	X =  49.000  mm,	Y =  112.000  mm,	Z =   -1.000 mm,
	W =-180.000 deg,	P =   0.000 deg,	R =    90.000 deg
};
P[5913]{
   GP1:
	UF : 1, UT : 4,		CONFIG : 'N U T, 0, 0, 0',
	X =  49.000  mm,	Y =  112.000  mm,	Z =   15.000 mm,
	W =-180.000 deg,	P =   0.000 deg,	R =    90.000 deg
};
P[5992]{
   GP1:
	UF : 1, UT : 4,		CONFIG : 'N U T, 0, 0, 0',
	X =  43.000  mm,	Y =  115.000  mm,	Z =   15.000 mm,
	W =-180.000 deg,	P =   0.000 deg,	R =    90.000 deg
};
P[5993]{
   GP1:
	UF : 1, UT : 4,		CONFIG : 'N U T, 0, 0, 0',
	X =  43.000  mm,	Y =  115.000  mm,	Z =   -1.000 mm,
	W =-180.000 deg,	P =   0.000 deg,	R =    90.000 deg
};
P[5994]{
   GP1:
	UF : 1, UT : 4,		CONFIG : 'N U T, 0, 0, 0',
	X =  43.000  mm,	Y =  115.000  mm,	Z =   15.000 mm,
	W =-180.000 deg,	P =   0.000 deg,	R =    90.000 deg
};
P[5995]{
   GP1:
	UF : 1, UT : 4,		CONFIG : 'N U T, 0, 0, 0',
	X =  46.000  mm,	Y =  115.000  mm,	Z =   15.000 mm,
	W =-180.000 deg,	P =   0.000 deg,	R =    90.000 deg
};
P[5996]{
   GP1:
	UF : 1, UT : 4,		CONFIG : 'N U T, 0, 0, 0',
	X =  46.000  mm,	Y =  115.000  mm,	Z =   -1.000 mm,
	W =-180.000 deg,	P =   0.000 deg,	R =    90.000 deg
};
P[5997]{
   GP1:
	UF : 1, UT : 4,		CONFIG : 'N U T, 0, 0, 0',
	X =  46.000  mm,	Y =  115.000  mm,	Z =   15.000 mm,
	W =-180.000 deg,	P =   0.000 deg,	R =    90.000 deg
};
P[5998]{
   GP1:
	UF : 1, UT : 4,		CONFIG : 'N U T, 0, 0, 0',
	X =  49.000  mm,	Y =  115.000  mm,	Z =   15.000 mm,
	W =-180.000 deg,	P =   0.000 deg,	R =    90.000 deg
};
P[5999]{
   GP1:
	UF : 1, UT : 4,		CONFIG : 'N U T, 0, 0, 0',
	X =  49.000  mm,	Y =  115.000  mm,	Z =   -1.000 mm,
	W =-180.000 deg,	P =   0.000 deg,	R =    90.000 deg
};
P[6000]{
   GP1:
	UF : 1, UT : 4,		CONFIG : 'N U T, 0, 0, 0',
	X =  49.000  mm,	Y =  115.000  mm,	Z =   15.000 mm,
	W =-180.000 deg,	P =   0.000 deg,	R =    90.000 deg
};
P[6001]{
   GP1:
	UF : 1, UT : 4,		CONFIG : 'N U T, 0, 0, 0',
	X =  52.000  mm,	Y =  115.000  mm,	Z =   15.000 mm,
	W =-180.000 deg,	P =   0.000 deg,	R =    90.000 deg
};
P[6002]{
   GP1:
	UF : 1, UT : 4,		CONFIG : 'N U T, 0, 0, 0',
	X =  52.000  mm,	Y =  115.000  mm,	Z =   -1.000 mm,
	W =-180.000 deg,	P =   0.000 deg,	R =    90.000 deg
};
P[6003]{
   GP1:
	UF : 1, UT : 4,		CONFIG : 'N U T, 0, 0, 0',
	X =  52.000  mm,	Y =  115.000  mm,	Z =   15.000 mm,
	W =-180.000 deg,	P =   0.000 deg,	R =    90.000 deg
};
P[6004]{
   GP1:
	UF : 1, UT : 4,		CONFIG : 'N U T, 0, 0, 0',
	X =  55.000  mm,	Y =  115.000  mm,	Z =   15.000 mm,
	W =-180.000 deg,	P =   0.000 deg,	R =    90.000 deg
};
P[6005]{
   GP1:
	UF : 1, UT : 4,		CONFIG : 'N U T, 0, 0, 0',
	X =  55.000  mm,	Y =  115.000  mm,	Z =   -1.000 mm,
	W =-180.000 deg,	P =   0.000 deg,	R =    90.000 deg
};
P[6006]{
   GP1:
	UF : 1, UT : 4,		CONFIG : 'N U T, 0, 0, 0',
	X =  55.000  mm,	Y =  115.000  mm,	Z =   15.000 mm,
	W =-180.000 deg,	P =   0.000 deg,	R =    90.000 deg
};
P[6007]{
   GP1:
	UF : 1, UT : 4,		CONFIG : 'N U T, 0, 0, 0',
	X =  58.000  mm,	Y =  115.000  mm,	Z =   15.000 mm,
	W =-180.000 deg,	P =   0.000 deg,	R =    90.000 deg
};
P[6008]{
   GP1:
	UF : 1, UT : 4,		CONFIG : 'N U T, 0, 0, 0',
	X =  58.000  mm,	Y =  115.000  mm,	Z =   -1.000 mm,
	W =-180.000 deg,	P =   0.000 deg,	R =    90.000 deg
};
P[6009]{
   GP1:
	UF : 1, UT : 4,		CONFIG : 'N U T, 0, 0, 0',
	X =  58.000  mm,	Y =  115.000  mm,	Z =   15.000 mm,
	W =-180.000 deg,	P =   0.000 deg,	R =    90.000 deg
};
P[6010]{
   GP1:
	UF : 1, UT : 4,		CONFIG : 'N U T, 0, 0, 0',
	X =  103.000  mm,	Y =  115.000  mm,	Z =   15.000 mm,
	W =-180.000 deg,	P =   0.000 deg,	R =    90.000 deg
};
P[6011]{
   GP1:
	UF : 1, UT : 4,		CONFIG : 'N U T, 0, 0, 0',
	X =  103.000  mm,	Y =  115.000  mm,	Z =   -1.000 mm,
	W =-180.000 deg,	P =   0.000 deg,	R =    90.000 deg
};
P[6012]{
   GP1:
	UF : 1, UT : 4,		CONFIG : 'N U T, 0, 0, 0',
	X =  103.000  mm,	Y =  115.000  mm,	Z =   15.000 mm,
	W =-180.000 deg,	P =   0.000 deg,	R =    90.000 deg
};
P[6058]{
   GP1:
	UF : 1, UT : 4,		CONFIG : 'N U T, 0, 0, 0',
	X =  16.000  mm,	Y =  118.000  mm,	Z =   15.000 mm,
	W =-180.000 deg,	P =   0.000 deg,	R =    90.000 deg
};
P[6059]{
   GP1:
	UF : 1, UT : 4,		CONFIG : 'N U T, 0, 0, 0',
	X =  16.000  mm,	Y =  118.000  mm,	Z =   -1.000 mm,
	W =-180.000 deg,	P =   0.000 deg,	R =    90.000 deg
};
P[6060]{
   GP1:
	UF : 1, UT : 4,		CONFIG : 'N U T, 0, 0, 0',
	X =  16.000  mm,	Y =  118.000  mm,	Z =   15.000 mm,
	W =-180.000 deg,	P =   0.000 deg,	R =    90.000 deg
};
P[6061]{
   GP1:
	UF : 1, UT : 4,		CONFIG : 'N U T, 0, 0, 0',
	X =  19.000  mm,	Y =  118.000  mm,	Z =   15.000 mm,
	W =-180.000 deg,	P =   0.000 deg,	R =    90.000 deg
};
P[6062]{
   GP1:
	UF : 1, UT : 4,		CONFIG : 'N U T, 0, 0, 0',
	X =  19.000  mm,	Y =  118.000  mm,	Z =   -1.000 mm,
	W =-180.000 deg,	P =   0.000 deg,	R =    90.000 deg
};
P[6063]{
   GP1:
	UF : 1, UT : 4,		CONFIG : 'N U T, 0, 0, 0',
	X =  19.000  mm,	Y =  118.000  mm,	Z =   15.000 mm,
	W =-180.000 deg,	P =   0.000 deg,	R =    90.000 deg
};
P[6070]{
   GP1:
	UF : 1, UT : 4,		CONFIG : 'N U T, 0, 0, 0',
	X =  28.000  mm,	Y =  118.000  mm,	Z =   15.000 mm,
	W =-180.000 deg,	P =   0.000 deg,	R =    90.000 deg
};
P[6071]{
   GP1:
	UF : 1, UT : 4,		CONFIG : 'N U T, 0, 0, 0',
	X =  28.000  mm,	Y =  118.000  mm,	Z =   -1.000 mm,
	W =-180.000 deg,	P =   0.000 deg,	R =    90.000 deg
};
P[6072]{
   GP1:
	UF : 1, UT : 4,		CONFIG : 'N U T, 0, 0, 0',
	X =  28.000  mm,	Y =  118.000  mm,	Z =   15.000 mm,
	W =-180.000 deg,	P =   0.000 deg,	R =    90.000 deg
};
P[6079]{
   GP1:
	UF : 1, UT : 4,		CONFIG : 'N U T, 0, 0, 0',
	X =  37.000  mm,	Y =  118.000  mm,	Z =   15.000 mm,
	W =-180.000 deg,	P =   0.000 deg,	R =    90.000 deg
};
P[6080]{
   GP1:
	UF : 1, UT : 4,		CONFIG : 'N U T, 0, 0, 0',
	X =  37.000  mm,	Y =  118.000  mm,	Z =   -1.000 mm,
	W =-180.000 deg,	P =   0.000 deg,	R =    90.000 deg
};
P[6081]{
   GP1:
	UF : 1, UT : 4,		CONFIG : 'N U T, 0, 0, 0',
	X =  37.000  mm,	Y =  118.000  mm,	Z =   15.000 mm,
	W =-180.000 deg,	P =   0.000 deg,	R =    90.000 deg
};
P[6082]{
   GP1:
	UF : 1, UT : 4,		CONFIG : 'N U T, 0, 0, 0',
	X =  40.000  mm,	Y =  118.000  mm,	Z =   15.000 mm,
	W =-180.000 deg,	P =   0.000 deg,	R =    90.000 deg
};
P[6083]{
   GP1:
	UF : 1, UT : 4,		CONFIG : 'N U T, 0, 0, 0',
	X =  40.000  mm,	Y =  118.000  mm,	Z =   -1.000 mm,
	W =-180.000 deg,	P =   0.000 deg,	R =    90.000 deg
};
P[6084]{
   GP1:
	UF : 1, UT : 4,		CONFIG : 'N U T, 0, 0, 0',
	X =  40.000  mm,	Y =  118.000  mm,	Z =   15.000 mm,
	W =-180.000 deg,	P =   0.000 deg,	R =    90.000 deg
};
P[6085]{
   GP1:
	UF : 1, UT : 4,		CONFIG : 'N U T, 0, 0, 0',
	X =  43.000  mm,	Y =  118.000  mm,	Z =   15.000 mm,
	W =-180.000 deg,	P =   0.000 deg,	R =    90.000 deg
};
P[6086]{
   GP1:
	UF : 1, UT : 4,		CONFIG : 'N U T, 0, 0, 0',
	X =  43.000  mm,	Y =  118.000  mm,	Z =   -1.000 mm,
	W =-180.000 deg,	P =   0.000 deg,	R =    90.000 deg
};
P[6087]{
   GP1:
	UF : 1, UT : 4,		CONFIG : 'N U T, 0, 0, 0',
	X =  43.000  mm,	Y =  118.000  mm,	Z =   15.000 mm,
	W =-180.000 deg,	P =   0.000 deg,	R =    90.000 deg
};
P[6088]{
   GP1:
	UF : 1, UT : 4,		CONFIG : 'N U T, 0, 0, 0',
	X =  46.000  mm,	Y =  118.000  mm,	Z =   15.000 mm,
	W =-180.000 deg,	P =   0.000 deg,	R =    90.000 deg
};
P[6089]{
   GP1:
	UF : 1, UT : 4,		CONFIG : 'N U T, 0, 0, 0',
	X =  46.000  mm,	Y =  118.000  mm,	Z =   -1.000 mm,
	W =-180.000 deg,	P =   0.000 deg,	R =    90.000 deg
};
P[6090]{
   GP1:
	UF : 1, UT : 4,		CONFIG : 'N U T, 0, 0, 0',
	X =  46.000  mm,	Y =  118.000  mm,	Z =   15.000 mm,
	W =-180.000 deg,	P =   0.000 deg,	R =    90.000 deg
};
P[6091]{
   GP1:
	UF : 1, UT : 4,		CONFIG : 'N U T, 0, 0, 0',
	X =  49.000  mm,	Y =  118.000  mm,	Z =   15.000 mm,
	W =-180.000 deg,	P =   0.000 deg,	R =    90.000 deg
};
P[6092]{
   GP1:
	UF : 1, UT : 4,		CONFIG : 'N U T, 0, 0, 0',
	X =  49.000  mm,	Y =  118.000  mm,	Z =   -1.000 mm,
	W =-180.000 deg,	P =   0.000 deg,	R =    90.000 deg
};
P[6093]{
   GP1:
	UF : 1, UT : 4,		CONFIG : 'N U T, 0, 0, 0',
	X =  49.000  mm,	Y =  118.000  mm,	Z =   15.000 mm,
	W =-180.000 deg,	P =   0.000 deg,	R =    90.000 deg
};
P[6094]{
   GP1:
	UF : 1, UT : 4,		CONFIG : 'N U T, 0, 0, 0',
	X =  52.000  mm,	Y =  118.000  mm,	Z =   15.000 mm,
	W =-180.000 deg,	P =   0.000 deg,	R =    90.000 deg
};
P[6095]{
   GP1:
	UF : 1, UT : 4,		CONFIG : 'N U T, 0, 0, 0',
	X =  52.000  mm,	Y =  118.000  mm,	Z =   -1.000 mm,
	W =-180.000 deg,	P =   0.000 deg,	R =    90.000 deg
};
P[6096]{
   GP1:
	UF : 1, UT : 4,		CONFIG : 'N U T, 0, 0, 0',
	X =  52.000  mm,	Y =  118.000  mm,	Z =   15.000 mm,
	W =-180.000 deg,	P =   0.000 deg,	R =    90.000 deg
};
P[6097]{
   GP1:
	UF : 1, UT : 4,		CONFIG : 'N U T, 0, 0, 0',
	X =  55.000  mm,	Y =  118.000  mm,	Z =   15.000 mm,
	W =-180.000 deg,	P =   0.000 deg,	R =    90.000 deg
};
P[6098]{
   GP1:
	UF : 1, UT : 4,		CONFIG : 'N U T, 0, 0, 0',
	X =  55.000  mm,	Y =  118.000  mm,	Z =   -1.000 mm,
	W =-180.000 deg,	P =   0.000 deg,	R =    90.000 deg
};
P[6099]{
   GP1:
	UF : 1, UT : 4,		CONFIG : 'N U T, 0, 0, 0',
	X =  55.000  mm,	Y =  118.000  mm,	Z =   15.000 mm,
	W =-180.000 deg,	P =   0.000 deg,	R =    90.000 deg
};
P[6100]{
   GP1:
	UF : 1, UT : 4,		CONFIG : 'N U T, 0, 0, 0',
	X =  58.000  mm,	Y =  118.000  mm,	Z =   15.000 mm,
	W =-180.000 deg,	P =   0.000 deg,	R =    90.000 deg
};
P[6101]{
   GP1:
	UF : 1, UT : 4,		CONFIG : 'N U T, 0, 0, 0',
	X =  58.000  mm,	Y =  118.000  mm,	Z =   -1.000 mm,
	W =-180.000 deg,	P =   0.000 deg,	R =    90.000 deg
};
P[6102]{
   GP1:
	UF : 1, UT : 4,		CONFIG : 'N U T, 0, 0, 0',
	X =  58.000  mm,	Y =  118.000  mm,	Z =   15.000 mm,
	W =-180.000 deg,	P =   0.000 deg,	R =    90.000 deg
};
P[6133]{
   GP1:
	UF : 1, UT : 4,		CONFIG : 'N U T, 0, 0, 0',
	X =  145.000  mm,	Y =  118.000  mm,	Z =   15.000 mm,
	W =-180.000 deg,	P =   0.000 deg,	R =    90.000 deg
};
P[6134]{
   GP1:
	UF : 1, UT : 4,		CONFIG : 'N U T, 0, 0, 0',
	X =  145.000  mm,	Y =  118.000  mm,	Z =   -1.000 mm,
	W =-180.000 deg,	P =   0.000 deg,	R =    90.000 deg
};
P[6135]{
   GP1:
	UF : 1, UT : 4,		CONFIG : 'N U T, 0, 0, 0',
	X =  145.000  mm,	Y =  118.000  mm,	Z =   15.000 mm,
	W =-180.000 deg,	P =   0.000 deg,	R =    90.000 deg
};
P[6160]{
   GP1:
	UF : 1, UT : 4,		CONFIG : 'N U T, 0, 0, 0',
	X =  16.000  mm,	Y =  121.000  mm,	Z =   15.000 mm,
	W =-180.000 deg,	P =   0.000 deg,	R =    90.000 deg
};
P[6161]{
   GP1:
	UF : 1, UT : 4,		CONFIG : 'N U T, 0, 0, 0',
	X =  16.000  mm,	Y =  121.000  mm,	Z =   -1.000 mm,
	W =-180.000 deg,	P =   0.000 deg,	R =    90.000 deg
};
P[6162]{
   GP1:
	UF : 1, UT : 4,		CONFIG : 'N U T, 0, 0, 0',
	X =  16.000  mm,	Y =  121.000  mm,	Z =   15.000 mm,
	W =-180.000 deg,	P =   0.000 deg,	R =    90.000 deg
};
P[6172]{
   GP1:
	UF : 1, UT : 4,		CONFIG : 'N U T, 0, 0, 0',
	X =  28.000  mm,	Y =  121.000  mm,	Z =   15.000 mm,
	W =-180.000 deg,	P =   0.000 deg,	R =    90.000 deg
};
P[6173]{
   GP1:
	UF : 1, UT : 4,		CONFIG : 'N U T, 0, 0, 0',
	X =  28.000  mm,	Y =  121.000  mm,	Z =   -1.000 mm,
	W =-180.000 deg,	P =   0.000 deg,	R =    90.000 deg
};
P[6174]{
   GP1:
	UF : 1, UT : 4,		CONFIG : 'N U T, 0, 0, 0',
	X =  28.000  mm,	Y =  121.000  mm,	Z =   15.000 mm,
	W =-180.000 deg,	P =   0.000 deg,	R =    90.000 deg
};
P[6187]{
   GP1:
	UF : 1, UT : 4,		CONFIG : 'N U T, 0, 0, 0',
	X =  43.000  mm,	Y =  121.000  mm,	Z =   15.000 mm,
	W =-180.000 deg,	P =   0.000 deg,	R =    90.000 deg
};
P[6188]{
   GP1:
	UF : 1, UT : 4,		CONFIG : 'N U T, 0, 0, 0',
	X =  43.000  mm,	Y =  121.000  mm,	Z =   -1.000 mm,
	W =-180.000 deg,	P =   0.000 deg,	R =    90.000 deg
};
P[6189]{
   GP1:
	UF : 1, UT : 4,		CONFIG : 'N U T, 0, 0, 0',
	X =  43.000  mm,	Y =  121.000  mm,	Z =   15.000 mm,
	W =-180.000 deg,	P =   0.000 deg,	R =    90.000 deg
};
P[6190]{
   GP1:
	UF : 1, UT : 4,		CONFIG : 'N U T, 0, 0, 0',
	X =  46.000  mm,	Y =  121.000  mm,	Z =   15.000 mm,
	W =-180.000 deg,	P =   0.000 deg,	R =    90.000 deg
};
P[6191]{
   GP1:
	UF : 1, UT : 4,		CONFIG : 'N U T, 0, 0, 0',
	X =  46.000  mm,	Y =  121.000  mm,	Z =   -1.000 mm,
	W =-180.000 deg,	P =   0.000 deg,	R =    90.000 deg
};
P[6192]{
   GP1:
	UF : 1, UT : 4,		CONFIG : 'N U T, 0, 0, 0',
	X =  46.000  mm,	Y =  121.000  mm,	Z =   15.000 mm,
	W =-180.000 deg,	P =   0.000 deg,	R =    90.000 deg
};
P[6193]{
   GP1:
	UF : 1, UT : 4,		CONFIG : 'N U T, 0, 0, 0',
	X =  49.000  mm,	Y =  121.000  mm,	Z =   15.000 mm,
	W =-180.000 deg,	P =   0.000 deg,	R =    90.000 deg
};
P[6194]{
   GP1:
	UF : 1, UT : 4,		CONFIG : 'N U T, 0, 0, 0',
	X =  49.000  mm,	Y =  121.000  mm,	Z =   -1.000 mm,
	W =-180.000 deg,	P =   0.000 deg,	R =    90.000 deg
};
P[6195]{
   GP1:
	UF : 1, UT : 4,		CONFIG : 'N U T, 0, 0, 0',
	X =  49.000  mm,	Y =  121.000  mm,	Z =   15.000 mm,
	W =-180.000 deg,	P =   0.000 deg,	R =    90.000 deg
};
P[6196]{
   GP1:
	UF : 1, UT : 4,		CONFIG : 'N U T, 0, 0, 0',
	X =  52.000  mm,	Y =  121.000  mm,	Z =   15.000 mm,
	W =-180.000 deg,	P =   0.000 deg,	R =    90.000 deg
};
P[6197]{
   GP1:
	UF : 1, UT : 4,		CONFIG : 'N U T, 0, 0, 0',
	X =  52.000  mm,	Y =  121.000  mm,	Z =   -1.000 mm,
	W =-180.000 deg,	P =   0.000 deg,	R =    90.000 deg
};
P[6198]{
   GP1:
	UF : 1, UT : 4,		CONFIG : 'N U T, 0, 0, 0',
	X =  52.000  mm,	Y =  121.000  mm,	Z =   15.000 mm,
	W =-180.000 deg,	P =   0.000 deg,	R =    90.000 deg
};
P[6199]{
   GP1:
	UF : 1, UT : 4,		CONFIG : 'N U T, 0, 0, 0',
	X =  55.000  mm,	Y =  121.000  mm,	Z =   15.000 mm,
	W =-180.000 deg,	P =   0.000 deg,	R =    90.000 deg
};
P[6200]{
   GP1:
	UF : 1, UT : 4,		CONFIG : 'N U T, 0, 0, 0',
	X =  55.000  mm,	Y =  121.000  mm,	Z =   -1.000 mm,
	W =-180.000 deg,	P =   0.000 deg,	R =    90.000 deg
};
P[6201]{
   GP1:
	UF : 1, UT : 4,		CONFIG : 'N U T, 0, 0, 0',
	X =  55.000  mm,	Y =  121.000  mm,	Z =   15.000 mm,
	W =-180.000 deg,	P =   0.000 deg,	R =    90.000 deg
};
P[6202]{
   GP1:
	UF : 1, UT : 4,		CONFIG : 'N U T, 0, 0, 0',
	X =  58.000  mm,	Y =  121.000  mm,	Z =   15.000 mm,
	W =-180.000 deg,	P =   0.000 deg,	R =    90.000 deg
};
P[6203]{
   GP1:
	UF : 1, UT : 4,		CONFIG : 'N U T, 0, 0, 0',
	X =  58.000  mm,	Y =  121.000  mm,	Z =   -1.000 mm,
	W =-180.000 deg,	P =   0.000 deg,	R =    90.000 deg
};
P[6204]{
   GP1:
	UF : 1, UT : 4,		CONFIG : 'N U T, 0, 0, 0',
	X =  58.000  mm,	Y =  121.000  mm,	Z =   15.000 mm,
	W =-180.000 deg,	P =   0.000 deg,	R =    90.000 deg
};
P[6205]{
   GP1:
	UF : 1, UT : 4,		CONFIG : 'N U T, 0, 0, 0',
	X =  61.000  mm,	Y =  121.000  mm,	Z =   15.000 mm,
	W =-180.000 deg,	P =   0.000 deg,	R =    90.000 deg
};
P[6206]{
   GP1:
	UF : 1, UT : 4,		CONFIG : 'N U T, 0, 0, 0',
	X =  61.000  mm,	Y =  121.000  mm,	Z =   -1.000 mm,
	W =-180.000 deg,	P =   0.000 deg,	R =    90.000 deg
};
P[6207]{
   GP1:
	UF : 1, UT : 4,		CONFIG : 'N U T, 0, 0, 0',
	X =  61.000  mm,	Y =  121.000  mm,	Z =   15.000 mm,
	W =-180.000 deg,	P =   0.000 deg,	R =    90.000 deg
};
P[6241]{
   GP1:
	UF : 1, UT : 4,		CONFIG : 'N U T, 0, 0, 0',
	X =  145.000  mm,	Y =  121.000  mm,	Z =   15.000 mm,
	W =-180.000 deg,	P =   0.000 deg,	R =    90.000 deg
};
P[6242]{
   GP1:
	UF : 1, UT : 4,		CONFIG : 'N U T, 0, 0, 0',
	X =  145.000  mm,	Y =  121.000  mm,	Z =   -1.000 mm,
	W =-180.000 deg,	P =   0.000 deg,	R =    90.000 deg
};
P[6243]{
   GP1:
	UF : 1, UT : 4,		CONFIG : 'N U T, 0, 0, 0',
	X =  145.000  mm,	Y =  121.000  mm,	Z =   15.000 mm,
	W =-180.000 deg,	P =   0.000 deg,	R =    90.000 deg
};
P[6244]{
   GP1:
	UF : 1, UT : 4,		CONFIG : 'N U T, 0, 0, 0',
	X =  148.000  mm,	Y =  121.000  mm,	Z =   15.000 mm,
	W =-180.000 deg,	P =   0.000 deg,	R =    90.000 deg
};
P[6245]{
   GP1:
	UF : 1, UT : 4,		CONFIG : 'N U T, 0, 0, 0',
	X =  148.000  mm,	Y =  121.000  mm,	Z =   -1.000 mm,
	W =-180.000 deg,	P =   0.000 deg,	R =    90.000 deg
};
P[6246]{
   GP1:
	UF : 1, UT : 4,		CONFIG : 'N U T, 0, 0, 0',
	X =  148.000  mm,	Y =  121.000  mm,	Z =   15.000 mm,
	W =-180.000 deg,	P =   0.000 deg,	R =    90.000 deg
};
P[6271]{
   GP1:
	UF : 1, UT : 4,		CONFIG : 'N U T, 0, 0, 0',
	X =  16.000  mm,	Y =  124.000  mm,	Z =   15.000 mm,
	W =-180.000 deg,	P =   0.000 deg,	R =    90.000 deg
};
P[6272]{
   GP1:
	UF : 1, UT : 4,		CONFIG : 'N U T, 0, 0, 0',
	X =  16.000  mm,	Y =  124.000  mm,	Z =   -1.000 mm,
	W =-180.000 deg,	P =   0.000 deg,	R =    90.000 deg
};
P[6273]{
   GP1:
	UF : 1, UT : 4,		CONFIG : 'N U T, 0, 0, 0',
	X =  16.000  mm,	Y =  124.000  mm,	Z =   15.000 mm,
	W =-180.000 deg,	P =   0.000 deg,	R =    90.000 deg
};
P[6274]{
   GP1:
	UF : 1, UT : 4,		CONFIG : 'N U T, 0, 0, 0',
	X =  19.000  mm,	Y =  124.000  mm,	Z =   15.000 mm,
	W =-180.000 deg,	P =   0.000 deg,	R =    90.000 deg
};
P[6275]{
   GP1:
	UF : 1, UT : 4,		CONFIG : 'N U T, 0, 0, 0',
	X =  19.000  mm,	Y =  124.000  mm,	Z =   -1.000 mm,
	W =-180.000 deg,	P =   0.000 deg,	R =    90.000 deg
};
P[6276]{
   GP1:
	UF : 1, UT : 4,		CONFIG : 'N U T, 0, 0, 0',
	X =  19.000  mm,	Y =  124.000  mm,	Z =   15.000 mm,
	W =-180.000 deg,	P =   0.000 deg,	R =    90.000 deg
};
P[6277]{
   GP1:
	UF : 1, UT : 4,		CONFIG : 'N U T, 0, 0, 0',
	X =  22.000  mm,	Y =  124.000  mm,	Z =   15.000 mm,
	W =-180.000 deg,	P =   0.000 deg,	R =    90.000 deg
};
P[6278]{
   GP1:
	UF : 1, UT : 4,		CONFIG : 'N U T, 0, 0, 0',
	X =  22.000  mm,	Y =  124.000  mm,	Z =   -1.000 mm,
	W =-180.000 deg,	P =   0.000 deg,	R =    90.000 deg
};
P[6279]{
   GP1:
	UF : 1, UT : 4,		CONFIG : 'N U T, 0, 0, 0',
	X =  22.000  mm,	Y =  124.000  mm,	Z =   15.000 mm,
	W =-180.000 deg,	P =   0.000 deg,	R =    90.000 deg
};
P[6283]{
   GP1:
	UF : 1, UT : 4,		CONFIG : 'N U T, 0, 0, 0',
	X =  28.000  mm,	Y =  124.000  mm,	Z =   15.000 mm,
	W =-180.000 deg,	P =   0.000 deg,	R =    90.000 deg
};
P[6284]{
   GP1:
	UF : 1, UT : 4,		CONFIG : 'N U T, 0, 0, 0',
	X =  28.000  mm,	Y =  124.000  mm,	Z =   -1.000 mm,
	W =-180.000 deg,	P =   0.000 deg,	R =    90.000 deg
};
P[6285]{
   GP1:
	UF : 1, UT : 4,		CONFIG : 'N U T, 0, 0, 0',
	X =  28.000  mm,	Y =  124.000  mm,	Z =   15.000 mm,
	W =-180.000 deg,	P =   0.000 deg,	R =    90.000 deg
};
P[6301]{
   GP1:
	UF : 1, UT : 4,		CONFIG : 'N U T, 0, 0, 0',
	X =  46.000  mm,	Y =  124.000  mm,	Z =   15.000 mm,
	W =-180.000 deg,	P =   0.000 deg,	R =    90.000 deg
};
P[6302]{
   GP1:
	UF : 1, UT : 4,		CONFIG : 'N U T, 0, 0, 0',
	X =  46.000  mm,	Y =  124.000  mm,	Z =   -1.000 mm,
	W =-180.000 deg,	P =   0.000 deg,	R =    90.000 deg
};
P[6303]{
   GP1:
	UF : 1, UT : 4,		CONFIG : 'N U T, 0, 0, 0',
	X =  46.000  mm,	Y =  124.000  mm,	Z =   15.000 mm,
	W =-180.000 deg,	P =   0.000 deg,	R =    90.000 deg
};
P[6304]{
   GP1:
	UF : 1, UT : 4,		CONFIG : 'N U T, 0, 0, 0',
	X =  49.000  mm,	Y =  124.000  mm,	Z =   15.000 mm,
	W =-180.000 deg,	P =   0.000 deg,	R =    90.000 deg
};
P[6305]{
   GP1:
	UF : 1, UT : 4,		CONFIG : 'N U T, 0, 0, 0',
	X =  49.000  mm,	Y =  124.000  mm,	Z =   -1.000 mm,
	W =-180.000 deg,	P =   0.000 deg,	R =    90.000 deg
};
P[6306]{
   GP1:
	UF : 1, UT : 4,		CONFIG : 'N U T, 0, 0, 0',
	X =  49.000  mm,	Y =  124.000  mm,	Z =   15.000 mm,
	W =-180.000 deg,	P =   0.000 deg,	R =    90.000 deg
};
P[6307]{
   GP1:
	UF : 1, UT : 4,		CONFIG : 'N U T, 0, 0, 0',
	X =  52.000  mm,	Y =  124.000  mm,	Z =   15.000 mm,
	W =-180.000 deg,	P =   0.000 deg,	R =    90.000 deg
};
P[6308]{
   GP1:
	UF : 1, UT : 4,		CONFIG : 'N U T, 0, 0, 0',
	X =  52.000  mm,	Y =  124.000  mm,	Z =   -1.000 mm,
	W =-180.000 deg,	P =   0.000 deg,	R =    90.000 deg
};
P[6309]{
   GP1:
	UF : 1, UT : 4,		CONFIG : 'N U T, 0, 0, 0',
	X =  52.000  mm,	Y =  124.000  mm,	Z =   15.000 mm,
	W =-180.000 deg,	P =   0.000 deg,	R =    90.000 deg
};
P[6310]{
   GP1:
	UF : 1, UT : 4,		CONFIG : 'N U T, 0, 0, 0',
	X =  55.000  mm,	Y =  124.000  mm,	Z =   15.000 mm,
	W =-180.000 deg,	P =   0.000 deg,	R =    90.000 deg
};
P[6311]{
   GP1:
	UF : 1, UT : 4,		CONFIG : 'N U T, 0, 0, 0',
	X =  55.000  mm,	Y =  124.000  mm,	Z =   -1.000 mm,
	W =-180.000 deg,	P =   0.000 deg,	R =    90.000 deg
};
P[6312]{
   GP1:
	UF : 1, UT : 4,		CONFIG : 'N U T, 0, 0, 0',
	X =  55.000  mm,	Y =  124.000  mm,	Z =   15.000 mm,
	W =-180.000 deg,	P =   0.000 deg,	R =    90.000 deg
};
P[6313]{
   GP1:
	UF : 1, UT : 4,		CONFIG : 'N U T, 0, 0, 0',
	X =  58.000  mm,	Y =  124.000  mm,	Z =   15.000 mm,
	W =-180.000 deg,	P =   0.000 deg,	R =    90.000 deg
};
P[6314]{
   GP1:
	UF : 1, UT : 4,		CONFIG : 'N U T, 0, 0, 0',
	X =  58.000  mm,	Y =  124.000  mm,	Z =   -1.000 mm,
	W =-180.000 deg,	P =   0.000 deg,	R =    90.000 deg
};
P[6315]{
   GP1:
	UF : 1, UT : 4,		CONFIG : 'N U T, 0, 0, 0',
	X =  58.000  mm,	Y =  124.000  mm,	Z =   15.000 mm,
	W =-180.000 deg,	P =   0.000 deg,	R =    90.000 deg
};
P[6316]{
   GP1:
	UF : 1, UT : 4,		CONFIG : 'N U T, 0, 0, 0',
	X =  61.000  mm,	Y =  124.000  mm,	Z =   15.000 mm,
	W =-180.000 deg,	P =   0.000 deg,	R =    90.000 deg
};
P[6317]{
   GP1:
	UF : 1, UT : 4,		CONFIG : 'N U T, 0, 0, 0',
	X =  61.000  mm,	Y =  124.000  mm,	Z =   -1.000 mm,
	W =-180.000 deg,	P =   0.000 deg,	R =    90.000 deg
};
P[6318]{
   GP1:
	UF : 1, UT : 4,		CONFIG : 'N U T, 0, 0, 0',
	X =  61.000  mm,	Y =  124.000  mm,	Z =   15.000 mm,
	W =-180.000 deg,	P =   0.000 deg,	R =    90.000 deg
};
P[6361]{
   GP1:
	UF : 1, UT : 4,		CONFIG : 'N U T, 0, 0, 0',
	X =  148.000  mm,	Y =  124.000  mm,	Z =   15.000 mm,
	W =-180.000 deg,	P =   0.000 deg,	R =    90.000 deg
};
P[6362]{
   GP1:
	UF : 1, UT : 4,		CONFIG : 'N U T, 0, 0, 0',
	X =  148.000  mm,	Y =  124.000  mm,	Z =   -1.000 mm,
	W =-180.000 deg,	P =   0.000 deg,	R =    90.000 deg
};
P[6363]{
   GP1:
	UF : 1, UT : 4,		CONFIG : 'N U T, 0, 0, 0',
	X =  148.000  mm,	Y =  124.000  mm,	Z =   15.000 mm,
	W =-180.000 deg,	P =   0.000 deg,	R =    90.000 deg
};
P[6379]{
   GP1:
	UF : 1, UT : 4,		CONFIG : 'N U T, 0, 0, 0',
	X =  16.000  mm,	Y =  127.000  mm,	Z =   15.000 mm,
	W =-180.000 deg,	P =   0.000 deg,	R =    90.000 deg
};
P[6380]{
   GP1:
	UF : 1, UT : 4,		CONFIG : 'N U T, 0, 0, 0',
	X =  16.000  mm,	Y =  127.000  mm,	Z =   -1.000 mm,
	W =-180.000 deg,	P =   0.000 deg,	R =    90.000 deg
};
P[6381]{
   GP1:
	UF : 1, UT : 4,		CONFIG : 'N U T, 0, 0, 0',
	X =  16.000  mm,	Y =  127.000  mm,	Z =   15.000 mm,
	W =-180.000 deg,	P =   0.000 deg,	R =    90.000 deg
};
P[6382]{
   GP1:
	UF : 1, UT : 4,		CONFIG : 'N U T, 0, 0, 0',
	X =  19.000  mm,	Y =  127.000  mm,	Z =   15.000 mm,
	W =-180.000 deg,	P =   0.000 deg,	R =    90.000 deg
};
P[6383]{
   GP1:
	UF : 1, UT : 4,		CONFIG : 'N U T, 0, 0, 0',
	X =  19.000  mm,	Y =  127.000  mm,	Z =   -1.000 mm,
	W =-180.000 deg,	P =   0.000 deg,	R =    90.000 deg
};
P[6384]{
   GP1:
	UF : 1, UT : 4,		CONFIG : 'N U T, 0, 0, 0',
	X =  19.000  mm,	Y =  127.000  mm,	Z =   15.000 mm,
	W =-180.000 deg,	P =   0.000 deg,	R =    90.000 deg
};
P[6385]{
   GP1:
	UF : 1, UT : 4,		CONFIG : 'N U T, 0, 0, 0',
	X =  22.000  mm,	Y =  127.000  mm,	Z =   15.000 mm,
	W =-180.000 deg,	P =   0.000 deg,	R =    90.000 deg
};
P[6386]{
   GP1:
	UF : 1, UT : 4,		CONFIG : 'N U T, 0, 0, 0',
	X =  22.000  mm,	Y =  127.000  mm,	Z =   -1.000 mm,
	W =-180.000 deg,	P =   0.000 deg,	R =    90.000 deg
};
P[6387]{
   GP1:
	UF : 1, UT : 4,		CONFIG : 'N U T, 0, 0, 0',
	X =  22.000  mm,	Y =  127.000  mm,	Z =   15.000 mm,
	W =-180.000 deg,	P =   0.000 deg,	R =    90.000 deg
};
P[6388]{
   GP1:
	UF : 1, UT : 4,		CONFIG : 'N U T, 0, 0, 0',
	X =  25.000  mm,	Y =  127.000  mm,	Z =   15.000 mm,
	W =-180.000 deg,	P =   0.000 deg,	R =    90.000 deg
};
P[6389]{
   GP1:
	UF : 1, UT : 4,		CONFIG : 'N U T, 0, 0, 0',
	X =  25.000  mm,	Y =  127.000  mm,	Z =   -1.000 mm,
	W =-180.000 deg,	P =   0.000 deg,	R =    90.000 deg
};
P[6390]{
   GP1:
	UF : 1, UT : 4,		CONFIG : 'N U T, 0, 0, 0',
	X =  25.000  mm,	Y =  127.000  mm,	Z =   15.000 mm,
	W =-180.000 deg,	P =   0.000 deg,	R =    90.000 deg
};
P[6391]{
   GP1:
	UF : 1, UT : 4,		CONFIG : 'N U T, 0, 0, 0',
	X =  28.000  mm,	Y =  127.000  mm,	Z =   15.000 mm,
	W =-180.000 deg,	P =   0.000 deg,	R =    90.000 deg
};
P[6392]{
   GP1:
	UF : 1, UT : 4,		CONFIG : 'N U T, 0, 0, 0',
	X =  28.000  mm,	Y =  127.000  mm,	Z =   -1.000 mm,
	W =-180.000 deg,	P =   0.000 deg,	R =    90.000 deg
};
P[6393]{
   GP1:
	UF : 1, UT : 4,		CONFIG : 'N U T, 0, 0, 0',
	X =  28.000  mm,	Y =  127.000  mm,	Z =   15.000 mm,
	W =-180.000 deg,	P =   0.000 deg,	R =    90.000 deg
};
P[6394]{
   GP1:
	UF : 1, UT : 4,		CONFIG : 'N U T, 0, 0, 0',
	X =  31.000  mm,	Y =  127.000  mm,	Z =   15.000 mm,
	W =-180.000 deg,	P =   0.000 deg,	R =    90.000 deg
};
P[6395]{
   GP1:
	UF : 1, UT : 4,		CONFIG : 'N U T, 0, 0, 0',
	X =  31.000  mm,	Y =  127.000  mm,	Z =   -1.000 mm,
	W =-180.000 deg,	P =   0.000 deg,	R =    90.000 deg
};
P[6396]{
   GP1:
	UF : 1, UT : 4,		CONFIG : 'N U T, 0, 0, 0',
	X =  31.000  mm,	Y =  127.000  mm,	Z =   15.000 mm,
	W =-180.000 deg,	P =   0.000 deg,	R =    90.000 deg
};
P[6397]{
   GP1:
	UF : 1, UT : 4,		CONFIG : 'N U T, 0, 0, 0',
	X =  34.000  mm,	Y =  127.000  mm,	Z =   15.000 mm,
	W =-180.000 deg,	P =   0.000 deg,	R =    90.000 deg
};
P[6398]{
   GP1:
	UF : 1, UT : 4,		CONFIG : 'N U T, 0, 0, 0',
	X =  34.000  mm,	Y =  127.000  mm,	Z =   -1.000 mm,
	W =-180.000 deg,	P =   0.000 deg,	R =    90.000 deg
};
P[6399]{
   GP1:
	UF : 1, UT : 4,		CONFIG : 'N U T, 0, 0, 0',
	X =  34.000  mm,	Y =  127.000  mm,	Z =   15.000 mm,
	W =-180.000 deg,	P =   0.000 deg,	R =    90.000 deg
};
P[6400]{
   GP1:
	UF : 1, UT : 4,		CONFIG : 'N U T, 0, 0, 0',
	X =  37.000  mm,	Y =  127.000  mm,	Z =   15.000 mm,
	W =-180.000 deg,	P =   0.000 deg,	R =    90.000 deg
};
P[6401]{
   GP1:
	UF : 1, UT : 4,		CONFIG : 'N U T, 0, 0, 0',
	X =  37.000  mm,	Y =  127.000  mm,	Z =   -1.000 mm,
	W =-180.000 deg,	P =   0.000 deg,	R =    90.000 deg
};
P[6402]{
   GP1:
	UF : 1, UT : 4,		CONFIG : 'N U T, 0, 0, 0',
	X =  37.000  mm,	Y =  127.000  mm,	Z =   15.000 mm,
	W =-180.000 deg,	P =   0.000 deg,	R =    90.000 deg
};
P[6403]{
   GP1:
	UF : 1, UT : 4,		CONFIG : 'N U T, 0, 0, 0',
	X =  40.000  mm,	Y =  127.000  mm,	Z =   15.000 mm,
	W =-180.000 deg,	P =   0.000 deg,	R =    90.000 deg
};
P[6404]{
   GP1:
	UF : 1, UT : 4,		CONFIG : 'N U T, 0, 0, 0',
	X =  40.000  mm,	Y =  127.000  mm,	Z =   -1.000 mm,
	W =-180.000 deg,	P =   0.000 deg,	R =    90.000 deg
};
P[6405]{
   GP1:
	UF : 1, UT : 4,		CONFIG : 'N U T, 0, 0, 0',
	X =  40.000  mm,	Y =  127.000  mm,	Z =   15.000 mm,
	W =-180.000 deg,	P =   0.000 deg,	R =    90.000 deg
};
P[6406]{
   GP1:
	UF : 1, UT : 4,		CONFIG : 'N U T, 0, 0, 0',
	X =  43.000  mm,	Y =  127.000  mm,	Z =   15.000 mm,
	W =-180.000 deg,	P =   0.000 deg,	R =    90.000 deg
};
P[6407]{
   GP1:
	UF : 1, UT : 4,		CONFIG : 'N U T, 0, 0, 0',
	X =  43.000  mm,	Y =  127.000  mm,	Z =   -1.000 mm,
	W =-180.000 deg,	P =   0.000 deg,	R =    90.000 deg
};
P[6408]{
   GP1:
	UF : 1, UT : 4,		CONFIG : 'N U T, 0, 0, 0',
	X =  43.000  mm,	Y =  127.000  mm,	Z =   15.000 mm,
	W =-180.000 deg,	P =   0.000 deg,	R =    90.000 deg
};
P[6409]{
   GP1:
	UF : 1, UT : 4,		CONFIG : 'N U T, 0, 0, 0',
	X =  46.000  mm,	Y =  127.000  mm,	Z =   15.000 mm,
	W =-180.000 deg,	P =   0.000 deg,	R =    90.000 deg
};
P[6410]{
   GP1:
	UF : 1, UT : 4,		CONFIG : 'N U T, 0, 0, 0',
	X =  46.000  mm,	Y =  127.000  mm,	Z =   -1.000 mm,
	W =-180.000 deg,	P =   0.000 deg,	R =    90.000 deg
};
P[6411]{
   GP1:
	UF : 1, UT : 4,		CONFIG : 'N U T, 0, 0, 0',
	X =  46.000  mm,	Y =  127.000  mm,	Z =   15.000 mm,
	W =-180.000 deg,	P =   0.000 deg,	R =    90.000 deg
};
P[6412]{
   GP1:
	UF : 1, UT : 4,		CONFIG : 'N U T, 0, 0, 0',
	X =  49.000  mm,	Y =  127.000  mm,	Z =   15.000 mm,
	W =-180.000 deg,	P =   0.000 deg,	R =    90.000 deg
};
P[6413]{
   GP1:
	UF : 1, UT : 4,		CONFIG : 'N U T, 0, 0, 0',
	X =  49.000  mm,	Y =  127.000  mm,	Z =   -1.000 mm,
	W =-180.000 deg,	P =   0.000 deg,	R =    90.000 deg
};
P[6414]{
   GP1:
	UF : 1, UT : 4,		CONFIG : 'N U T, 0, 0, 0',
	X =  49.000  mm,	Y =  127.000  mm,	Z =   15.000 mm,
	W =-180.000 deg,	P =   0.000 deg,	R =    90.000 deg
};
P[6415]{
   GP1:
	UF : 1, UT : 4,		CONFIG : 'N U T, 0, 0, 0',
	X =  52.000  mm,	Y =  127.000  mm,	Z =   15.000 mm,
	W =-180.000 deg,	P =   0.000 deg,	R =    90.000 deg
};
P[6416]{
   GP1:
	UF : 1, UT : 4,		CONFIG : 'N U T, 0, 0, 0',
	X =  52.000  mm,	Y =  127.000  mm,	Z =   -1.000 mm,
	W =-180.000 deg,	P =   0.000 deg,	R =    90.000 deg
};
P[6417]{
   GP1:
	UF : 1, UT : 4,		CONFIG : 'N U T, 0, 0, 0',
	X =  52.000  mm,	Y =  127.000  mm,	Z =   15.000 mm,
	W =-180.000 deg,	P =   0.000 deg,	R =    90.000 deg
};
P[6418]{
   GP1:
	UF : 1, UT : 4,		CONFIG : 'N U T, 0, 0, 0',
	X =  55.000  mm,	Y =  127.000  mm,	Z =   15.000 mm,
	W =-180.000 deg,	P =   0.000 deg,	R =    90.000 deg
};
P[6419]{
   GP1:
	UF : 1, UT : 4,		CONFIG : 'N U T, 0, 0, 0',
	X =  55.000  mm,	Y =  127.000  mm,	Z =   -1.000 mm,
	W =-180.000 deg,	P =   0.000 deg,	R =    90.000 deg
};
P[6420]{
   GP1:
	UF : 1, UT : 4,		CONFIG : 'N U T, 0, 0, 0',
	X =  55.000  mm,	Y =  127.000  mm,	Z =   15.000 mm,
	W =-180.000 deg,	P =   0.000 deg,	R =    90.000 deg
};
P[6421]{
   GP1:
	UF : 1, UT : 4,		CONFIG : 'N U T, 0, 0, 0',
	X =  58.000  mm,	Y =  127.000  mm,	Z =   15.000 mm,
	W =-180.000 deg,	P =   0.000 deg,	R =    90.000 deg
};
P[6422]{
   GP1:
	UF : 1, UT : 4,		CONFIG : 'N U T, 0, 0, 0',
	X =  58.000  mm,	Y =  127.000  mm,	Z =   -1.000 mm,
	W =-180.000 deg,	P =   0.000 deg,	R =    90.000 deg
};
P[6423]{
   GP1:
	UF : 1, UT : 4,		CONFIG : 'N U T, 0, 0, 0',
	X =  58.000  mm,	Y =  127.000  mm,	Z =   15.000 mm,
	W =-180.000 deg,	P =   0.000 deg,	R =    90.000 deg
};
P[6424]{
   GP1:
	UF : 1, UT : 4,		CONFIG : 'N U T, 0, 0, 0',
	X =  61.000  mm,	Y =  127.000  mm,	Z =   15.000 mm,
	W =-180.000 deg,	P =   0.000 deg,	R =    90.000 deg
};
P[6425]{
   GP1:
	UF : 1, UT : 4,		CONFIG : 'N U T, 0, 0, 0',
	X =  61.000  mm,	Y =  127.000  mm,	Z =   -1.000 mm,
	W =-180.000 deg,	P =   0.000 deg,	R =    90.000 deg
};
P[6426]{
   GP1:
	UF : 1, UT : 4,		CONFIG : 'N U T, 0, 0, 0',
	X =  61.000  mm,	Y =  127.000  mm,	Z =   15.000 mm,
	W =-180.000 deg,	P =   0.000 deg,	R =    90.000 deg
};
P[6505]{
   GP1:
	UF : 1, UT : 4,		CONFIG : 'N U T, 0, 0, 0',
	X =  16.000  mm,	Y =  130.000  mm,	Z =   15.000 mm,
	W =-180.000 deg,	P =   0.000 deg,	R =    90.000 deg
};
P[6506]{
   GP1:
	UF : 1, UT : 4,		CONFIG : 'N U T, 0, 0, 0',
	X =  16.000  mm,	Y =  130.000  mm,	Z =   -1.000 mm,
	W =-180.000 deg,	P =   0.000 deg,	R =    90.000 deg
};
P[6507]{
   GP1:
	UF : 1, UT : 4,		CONFIG : 'N U T, 0, 0, 0',
	X =  16.000  mm,	Y =  130.000  mm,	Z =   15.000 mm,
	W =-180.000 deg,	P =   0.000 deg,	R =    90.000 deg
};
P[6508]{
   GP1:
	UF : 1, UT : 4,		CONFIG : 'N U T, 0, 0, 0',
	X =  19.000  mm,	Y =  130.000  mm,	Z =   15.000 mm,
	W =-180.000 deg,	P =   0.000 deg,	R =    90.000 deg
};
P[6509]{
   GP1:
	UF : 1, UT : 4,		CONFIG : 'N U T, 0, 0, 0',
	X =  19.000  mm,	Y =  130.000  mm,	Z =   -1.000 mm,
	W =-180.000 deg,	P =   0.000 deg,	R =    90.000 deg
};
P[6510]{
   GP1:
	UF : 1, UT : 4,		CONFIG : 'N U T, 0, 0, 0',
	X =  19.000  mm,	Y =  130.000  mm,	Z =   15.000 mm,
	W =-180.000 deg,	P =   0.000 deg,	R =    90.000 deg
};
P[6511]{
   GP1:
	UF : 1, UT : 4,		CONFIG : 'N U T, 0, 0, 0',
	X =  22.000  mm,	Y =  130.000  mm,	Z =   15.000 mm,
	W =-180.000 deg,	P =   0.000 deg,	R =    90.000 deg
};
P[6512]{
   GP1:
	UF : 1, UT : 4,		CONFIG : 'N U T, 0, 0, 0',
	X =  22.000  mm,	Y =  130.000  mm,	Z =   -1.000 mm,
	W =-180.000 deg,	P =   0.000 deg,	R =    90.000 deg
};
P[6513]{
   GP1:
	UF : 1, UT : 4,		CONFIG : 'N U T, 0, 0, 0',
	X =  22.000  mm,	Y =  130.000  mm,	Z =   15.000 mm,
	W =-180.000 deg,	P =   0.000 deg,	R =    90.000 deg
};
P[6514]{
   GP1:
	UF : 1, UT : 4,		CONFIG : 'N U T, 0, 0, 0',
	X =  25.000  mm,	Y =  130.000  mm,	Z =   15.000 mm,
	W =-180.000 deg,	P =   0.000 deg,	R =    90.000 deg
};
P[6515]{
   GP1:
	UF : 1, UT : 4,		CONFIG : 'N U T, 0, 0, 0',
	X =  25.000  mm,	Y =  130.000  mm,	Z =   -1.000 mm,
	W =-180.000 deg,	P =   0.000 deg,	R =    90.000 deg
};
P[6516]{
   GP1:
	UF : 1, UT : 4,		CONFIG : 'N U T, 0, 0, 0',
	X =  25.000  mm,	Y =  130.000  mm,	Z =   15.000 mm,
	W =-180.000 deg,	P =   0.000 deg,	R =    90.000 deg
};
P[6517]{
   GP1:
	UF : 1, UT : 4,		CONFIG : 'N U T, 0, 0, 0',
	X =  28.000  mm,	Y =  130.000  mm,	Z =   15.000 mm,
	W =-180.000 deg,	P =   0.000 deg,	R =    90.000 deg
};
P[6518]{
   GP1:
	UF : 1, UT : 4,		CONFIG : 'N U T, 0, 0, 0',
	X =  28.000  mm,	Y =  130.000  mm,	Z =   -1.000 mm,
	W =-180.000 deg,	P =   0.000 deg,	R =    90.000 deg
};
P[6519]{
   GP1:
	UF : 1, UT : 4,		CONFIG : 'N U T, 0, 0, 0',
	X =  28.000  mm,	Y =  130.000  mm,	Z =   15.000 mm,
	W =-180.000 deg,	P =   0.000 deg,	R =    90.000 deg
};
P[6520]{
   GP1:
	UF : 1, UT : 4,		CONFIG : 'N U T, 0, 0, 0',
	X =  31.000  mm,	Y =  130.000  mm,	Z =   15.000 mm,
	W =-180.000 deg,	P =   0.000 deg,	R =    90.000 deg
};
P[6521]{
   GP1:
	UF : 1, UT : 4,		CONFIG : 'N U T, 0, 0, 0',
	X =  31.000  mm,	Y =  130.000  mm,	Z =   -1.000 mm,
	W =-180.000 deg,	P =   0.000 deg,	R =    90.000 deg
};
P[6522]{
   GP1:
	UF : 1, UT : 4,		CONFIG : 'N U T, 0, 0, 0',
	X =  31.000  mm,	Y =  130.000  mm,	Z =   15.000 mm,
	W =-180.000 deg,	P =   0.000 deg,	R =    90.000 deg
};
P[6523]{
   GP1:
	UF : 1, UT : 4,		CONFIG : 'N U T, 0, 0, 0',
	X =  34.000  mm,	Y =  130.000  mm,	Z =   15.000 mm,
	W =-180.000 deg,	P =   0.000 deg,	R =    90.000 deg
};
P[6524]{
   GP1:
	UF : 1, UT : 4,		CONFIG : 'N U T, 0, 0, 0',
	X =  34.000  mm,	Y =  130.000  mm,	Z =   -1.000 mm,
	W =-180.000 deg,	P =   0.000 deg,	R =    90.000 deg
};
P[6525]{
   GP1:
	UF : 1, UT : 4,		CONFIG : 'N U T, 0, 0, 0',
	X =  34.000  mm,	Y =  130.000  mm,	Z =   15.000 mm,
	W =-180.000 deg,	P =   0.000 deg,	R =    90.000 deg
};
P[6526]{
   GP1:
	UF : 1, UT : 4,		CONFIG : 'N U T, 0, 0, 0',
	X =  40.000  mm,	Y =  130.000  mm,	Z =   15.000 mm,
	W =-180.000 deg,	P =   0.000 deg,	R =    90.000 deg
};
P[6527]{
   GP1:
	UF : 1, UT : 4,		CONFIG : 'N U T, 0, 0, 0',
	X =  40.000  mm,	Y =  130.000  mm,	Z =   -1.000 mm,
	W =-180.000 deg,	P =   0.000 deg,	R =    90.000 deg
};
P[6528]{
   GP1:
	UF : 1, UT : 4,		CONFIG : 'N U T, 0, 0, 0',
	X =  40.000  mm,	Y =  130.000  mm,	Z =   15.000 mm,
	W =-180.000 deg,	P =   0.000 deg,	R =    90.000 deg
};
P[6529]{
   GP1:
	UF : 1, UT : 4,		CONFIG : 'N U T, 0, 0, 0',
	X =  43.000  mm,	Y =  130.000  mm,	Z =   15.000 mm,
	W =-180.000 deg,	P =   0.000 deg,	R =    90.000 deg
};
P[6530]{
   GP1:
	UF : 1, UT : 4,		CONFIG : 'N U T, 0, 0, 0',
	X =  43.000  mm,	Y =  130.000  mm,	Z =   -1.000 mm,
	W =-180.000 deg,	P =   0.000 deg,	R =    90.000 deg
};
P[6531]{
   GP1:
	UF : 1, UT : 4,		CONFIG : 'N U T, 0, 0, 0',
	X =  43.000  mm,	Y =  130.000  mm,	Z =   15.000 mm,
	W =-180.000 deg,	P =   0.000 deg,	R =    90.000 deg
};
P[6532]{
   GP1:
	UF : 1, UT : 4,		CONFIG : 'N U T, 0, 0, 0',
	X =  46.000  mm,	Y =  130.000  mm,	Z =   15.000 mm,
	W =-180.000 deg,	P =   0.000 deg,	R =    90.000 deg
};
P[6533]{
   GP1:
	UF : 1, UT : 4,		CONFIG : 'N U T, 0, 0, 0',
	X =  46.000  mm,	Y =  130.000  mm,	Z =   -1.000 mm,
	W =-180.000 deg,	P =   0.000 deg,	R =    90.000 deg
};
P[6534]{
   GP1:
	UF : 1, UT : 4,		CONFIG : 'N U T, 0, 0, 0',
	X =  46.000  mm,	Y =  130.000  mm,	Z =   15.000 mm,
	W =-180.000 deg,	P =   0.000 deg,	R =    90.000 deg
};
P[6535]{
   GP1:
	UF : 1, UT : 4,		CONFIG : 'N U T, 0, 0, 0',
	X =  49.000  mm,	Y =  130.000  mm,	Z =   15.000 mm,
	W =-180.000 deg,	P =   0.000 deg,	R =    90.000 deg
};
P[6536]{
   GP1:
	UF : 1, UT : 4,		CONFIG : 'N U T, 0, 0, 0',
	X =  49.000  mm,	Y =  130.000  mm,	Z =   -1.000 mm,
	W =-180.000 deg,	P =   0.000 deg,	R =    90.000 deg
};
P[6537]{
   GP1:
	UF : 1, UT : 4,		CONFIG : 'N U T, 0, 0, 0',
	X =  49.000  mm,	Y =  130.000  mm,	Z =   15.000 mm,
	W =-180.000 deg,	P =   0.000 deg,	R =    90.000 deg
};
P[6538]{
   GP1:
	UF : 1, UT : 4,		CONFIG : 'N U T, 0, 0, 0',
	X =  52.000  mm,	Y =  130.000  mm,	Z =   15.000 mm,
	W =-180.000 deg,	P =   0.000 deg,	R =    90.000 deg
};
P[6539]{
   GP1:
	UF : 1, UT : 4,		CONFIG : 'N U T, 0, 0, 0',
	X =  52.000  mm,	Y =  130.000  mm,	Z =   -1.000 mm,
	W =-180.000 deg,	P =   0.000 deg,	R =    90.000 deg
};
P[6540]{
   GP1:
	UF : 1, UT : 4,		CONFIG : 'N U T, 0, 0, 0',
	X =  52.000  mm,	Y =  130.000  mm,	Z =   15.000 mm,
	W =-180.000 deg,	P =   0.000 deg,	R =    90.000 deg
};
P[6541]{
   GP1:
	UF : 1, UT : 4,		CONFIG : 'N U T, 0, 0, 0',
	X =  55.000  mm,	Y =  130.000  mm,	Z =   15.000 mm,
	W =-180.000 deg,	P =   0.000 deg,	R =    90.000 deg
};
P[6542]{
   GP1:
	UF : 1, UT : 4,		CONFIG : 'N U T, 0, 0, 0',
	X =  55.000  mm,	Y =  130.000  mm,	Z =   -1.000 mm,
	W =-180.000 deg,	P =   0.000 deg,	R =    90.000 deg
};
P[6543]{
   GP1:
	UF : 1, UT : 4,		CONFIG : 'N U T, 0, 0, 0',
	X =  55.000  mm,	Y =  130.000  mm,	Z =   15.000 mm,
	W =-180.000 deg,	P =   0.000 deg,	R =    90.000 deg
};
P[6544]{
   GP1:
	UF : 1, UT : 4,		CONFIG : 'N U T, 0, 0, 0',
	X =  58.000  mm,	Y =  130.000  mm,	Z =   15.000 mm,
	W =-180.000 deg,	P =   0.000 deg,	R =    90.000 deg
};
P[6545]{
   GP1:
	UF : 1, UT : 4,		CONFIG : 'N U T, 0, 0, 0',
	X =  58.000  mm,	Y =  130.000  mm,	Z =   -1.000 mm,
	W =-180.000 deg,	P =   0.000 deg,	R =    90.000 deg
};
P[6546]{
   GP1:
	UF : 1, UT : 4,		CONFIG : 'N U T, 0, 0, 0',
	X =  58.000  mm,	Y =  130.000  mm,	Z =   15.000 mm,
	W =-180.000 deg,	P =   0.000 deg,	R =    90.000 deg
};
P[6547]{
   GP1:
	UF : 1, UT : 4,		CONFIG : 'N U T, 0, 0, 0',
	X =  61.000  mm,	Y =  130.000  mm,	Z =   15.000 mm,
	W =-180.000 deg,	P =   0.000 deg,	R =    90.000 deg
};
P[6548]{
   GP1:
	UF : 1, UT : 4,		CONFIG : 'N U T, 0, 0, 0',
	X =  61.000  mm,	Y =  130.000  mm,	Z =   -1.000 mm,
	W =-180.000 deg,	P =   0.000 deg,	R =    90.000 deg
};
P[6549]{
   GP1:
	UF : 1, UT : 4,		CONFIG : 'N U T, 0, 0, 0',
	X =  61.000  mm,	Y =  130.000  mm,	Z =   15.000 mm,
	W =-180.000 deg,	P =   0.000 deg,	R =    90.000 deg
};
P[6595]{
   GP1:
	UF : 1, UT : 4,		CONFIG : 'N U T, 0, 0, 0',
	X =  151.000  mm,	Y =  130.000  mm,	Z =   15.000 mm,
	W =-180.000 deg,	P =   0.000 deg,	R =    90.000 deg
};
P[6596]{
   GP1:
	UF : 1, UT : 4,		CONFIG : 'N U T, 0, 0, 0',
	X =  151.000  mm,	Y =  130.000  mm,	Z =   -1.000 mm,
	W =-180.000 deg,	P =   0.000 deg,	R =    90.000 deg
};
P[6597]{
   GP1:
	UF : 1, UT : 4,		CONFIG : 'N U T, 0, 0, 0',
	X =  151.000  mm,	Y =  130.000  mm,	Z =   15.000 mm,
	W =-180.000 deg,	P =   0.000 deg,	R =    90.000 deg
};
P[6622]{
   GP1:
	UF : 1, UT : 4,		CONFIG : 'N U T, 0, 0, 0',
	X =  16.000  mm,	Y =  133.000  mm,	Z =   15.000 mm,
	W =-180.000 deg,	P =   0.000 deg,	R =    90.000 deg
};
P[6623]{
   GP1:
	UF : 1, UT : 4,		CONFIG : 'N U T, 0, 0, 0',
	X =  16.000  mm,	Y =  133.000  mm,	Z =   -1.000 mm,
	W =-180.000 deg,	P =   0.000 deg,	R =    90.000 deg
};
P[6624]{
   GP1:
	UF : 1, UT : 4,		CONFIG : 'N U T, 0, 0, 0',
	X =  16.000  mm,	Y =  133.000  mm,	Z =   15.000 mm,
	W =-180.000 deg,	P =   0.000 deg,	R =    90.000 deg
};
P[6625]{
   GP1:
	UF : 1, UT : 4,		CONFIG : 'N U T, 0, 0, 0',
	X =  19.000  mm,	Y =  133.000  mm,	Z =   15.000 mm,
	W =-180.000 deg,	P =   0.000 deg,	R =    90.000 deg
};
P[6626]{
   GP1:
	UF : 1, UT : 4,		CONFIG : 'N U T, 0, 0, 0',
	X =  19.000  mm,	Y =  133.000  mm,	Z =   -1.000 mm,
	W =-180.000 deg,	P =   0.000 deg,	R =    90.000 deg
};
P[6627]{
   GP1:
	UF : 1, UT : 4,		CONFIG : 'N U T, 0, 0, 0',
	X =  19.000  mm,	Y =  133.000  mm,	Z =   15.000 mm,
	W =-180.000 deg,	P =   0.000 deg,	R =    90.000 deg
};
P[6628]{
   GP1:
	UF : 1, UT : 4,		CONFIG : 'N U T, 0, 0, 0',
	X =  22.000  mm,	Y =  133.000  mm,	Z =   15.000 mm,
	W =-180.000 deg,	P =   0.000 deg,	R =    90.000 deg
};
P[6629]{
   GP1:
	UF : 1, UT : 4,		CONFIG : 'N U T, 0, 0, 0',
	X =  22.000  mm,	Y =  133.000  mm,	Z =   -1.000 mm,
	W =-180.000 deg,	P =   0.000 deg,	R =    90.000 deg
};
P[6630]{
   GP1:
	UF : 1, UT : 4,		CONFIG : 'N U T, 0, 0, 0',
	X =  22.000  mm,	Y =  133.000  mm,	Z =   15.000 mm,
	W =-180.000 deg,	P =   0.000 deg,	R =    90.000 deg
};
P[6631]{
   GP1:
	UF : 1, UT : 4,		CONFIG : 'N U T, 0, 0, 0',
	X =  25.000  mm,	Y =  133.000  mm,	Z =   15.000 mm,
	W =-180.000 deg,	P =   0.000 deg,	R =    90.000 deg
};
P[6632]{
   GP1:
	UF : 1, UT : 4,		CONFIG : 'N U T, 0, 0, 0',
	X =  25.000  mm,	Y =  133.000  mm,	Z =   -1.000 mm,
	W =-180.000 deg,	P =   0.000 deg,	R =    90.000 deg
};
P[6633]{
   GP1:
	UF : 1, UT : 4,		CONFIG : 'N U T, 0, 0, 0',
	X =  25.000  mm,	Y =  133.000  mm,	Z =   15.000 mm,
	W =-180.000 deg,	P =   0.000 deg,	R =    90.000 deg
};
P[6634]{
   GP1:
	UF : 1, UT : 4,		CONFIG : 'N U T, 0, 0, 0',
	X =  28.000  mm,	Y =  133.000  mm,	Z =   15.000 mm,
	W =-180.000 deg,	P =   0.000 deg,	R =    90.000 deg
};
P[6635]{
   GP1:
	UF : 1, UT : 4,		CONFIG : 'N U T, 0, 0, 0',
	X =  28.000  mm,	Y =  133.000  mm,	Z =   -1.000 mm,
	W =-180.000 deg,	P =   0.000 deg,	R =    90.000 deg
};
P[6636]{
   GP1:
	UF : 1, UT : 4,		CONFIG : 'N U T, 0, 0, 0',
	X =  28.000  mm,	Y =  133.000  mm,	Z =   15.000 mm,
	W =-180.000 deg,	P =   0.000 deg,	R =    90.000 deg
};
P[6637]{
   GP1:
	UF : 1, UT : 4,		CONFIG : 'N U T, 0, 0, 0',
	X =  31.000  mm,	Y =  133.000  mm,	Z =   15.000 mm,
	W =-180.000 deg,	P =   0.000 deg,	R =    90.000 deg
};
P[6638]{
   GP1:
	UF : 1, UT : 4,		CONFIG : 'N U T, 0, 0, 0',
	X =  31.000  mm,	Y =  133.000  mm,	Z =   -1.000 mm,
	W =-180.000 deg,	P =   0.000 deg,	R =    90.000 deg
};
P[6639]{
   GP1:
	UF : 1, UT : 4,		CONFIG : 'N U T, 0, 0, 0',
	X =  31.000  mm,	Y =  133.000  mm,	Z =   15.000 mm,
	W =-180.000 deg,	P =   0.000 deg,	R =    90.000 deg
};
P[6640]{
   GP1:
	UF : 1, UT : 4,		CONFIG : 'N U T, 0, 0, 0',
	X =  34.000  mm,	Y =  133.000  mm,	Z =   15.000 mm,
	W =-180.000 deg,	P =   0.000 deg,	R =    90.000 deg
};
P[6641]{
   GP1:
	UF : 1, UT : 4,		CONFIG : 'N U T, 0, 0, 0',
	X =  34.000  mm,	Y =  133.000  mm,	Z =   -1.000 mm,
	W =-180.000 deg,	P =   0.000 deg,	R =    90.000 deg
};
P[6642]{
   GP1:
	UF : 1, UT : 4,		CONFIG : 'N U T, 0, 0, 0',
	X =  34.000  mm,	Y =  133.000  mm,	Z =   15.000 mm,
	W =-180.000 deg,	P =   0.000 deg,	R =    90.000 deg
};
P[6643]{
   GP1:
	UF : 1, UT : 4,		CONFIG : 'N U T, 0, 0, 0',
	X =  37.000  mm,	Y =  133.000  mm,	Z =   15.000 mm,
	W =-180.000 deg,	P =   0.000 deg,	R =    90.000 deg
};
P[6644]{
   GP1:
	UF : 1, UT : 4,		CONFIG : 'N U T, 0, 0, 0',
	X =  37.000  mm,	Y =  133.000  mm,	Z =   -1.000 mm,
	W =-180.000 deg,	P =   0.000 deg,	R =    90.000 deg
};
P[6645]{
   GP1:
	UF : 1, UT : 4,		CONFIG : 'N U T, 0, 0, 0',
	X =  37.000  mm,	Y =  133.000  mm,	Z =   15.000 mm,
	W =-180.000 deg,	P =   0.000 deg,	R =    90.000 deg
};
P[6646]{
   GP1:
	UF : 1, UT : 4,		CONFIG : 'N U T, 0, 0, 0',
	X =  40.000  mm,	Y =  133.000  mm,	Z =   15.000 mm,
	W =-180.000 deg,	P =   0.000 deg,	R =    90.000 deg
};
P[6647]{
   GP1:
	UF : 1, UT : 4,		CONFIG : 'N U T, 0, 0, 0',
	X =  40.000  mm,	Y =  133.000  mm,	Z =   -1.000 mm,
	W =-180.000 deg,	P =   0.000 deg,	R =    90.000 deg
};
P[6648]{
   GP1:
	UF : 1, UT : 4,		CONFIG : 'N U T, 0, 0, 0',
	X =  40.000  mm,	Y =  133.000  mm,	Z =   15.000 mm,
	W =-180.000 deg,	P =   0.000 deg,	R =    90.000 deg
};
P[6649]{
   GP1:
	UF : 1, UT : 4,		CONFIG : 'N U T, 0, 0, 0',
	X =  43.000  mm,	Y =  133.000  mm,	Z =   15.000 mm,
	W =-180.000 deg,	P =   0.000 deg,	R =    90.000 deg
};
P[6650]{
   GP1:
	UF : 1, UT : 4,		CONFIG : 'N U T, 0, 0, 0',
	X =  43.000  mm,	Y =  133.000  mm,	Z =   -1.000 mm,
	W =-180.000 deg,	P =   0.000 deg,	R =    90.000 deg
};
P[6651]{
   GP1:
	UF : 1, UT : 4,		CONFIG : 'N U T, 0, 0, 0',
	X =  43.000  mm,	Y =  133.000  mm,	Z =   15.000 mm,
	W =-180.000 deg,	P =   0.000 deg,	R =    90.000 deg
};
P[6667]{
   GP1:
	UF : 1, UT : 4,		CONFIG : 'N U T, 0, 0, 0',
	X =  61.000  mm,	Y =  133.000  mm,	Z =   15.000 mm,
	W =-180.000 deg,	P =   0.000 deg,	R =    90.000 deg
};
P[6668]{
   GP1:
	UF : 1, UT : 4,		CONFIG : 'N U T, 0, 0, 0',
	X =  61.000  mm,	Y =  133.000  mm,	Z =   -1.000 mm,
	W =-180.000 deg,	P =   0.000 deg,	R =    90.000 deg
};
P[6669]{
   GP1:
	UF : 1, UT : 4,		CONFIG : 'N U T, 0, 0, 0',
	X =  61.000  mm,	Y =  133.000  mm,	Z =   15.000 mm,
	W =-180.000 deg,	P =   0.000 deg,	R =    90.000 deg
};
P[6673]{
   GP1:
	UF : 1, UT : 4,		CONFIG : 'N U T, 0, 0, 0',
	X =  67.000  mm,	Y =  133.000  mm,	Z =   15.000 mm,
	W =-180.000 deg,	P =   0.000 deg,	R =    90.000 deg
};
P[6674]{
   GP1:
	UF : 1, UT : 4,		CONFIG : 'N U T, 0, 0, 0',
	X =  67.000  mm,	Y =  133.000  mm,	Z =   -1.000 mm,
	W =-180.000 deg,	P =   0.000 deg,	R =    90.000 deg
};
P[6675]{
   GP1:
	UF : 1, UT : 4,		CONFIG : 'N U T, 0, 0, 0',
	X =  67.000  mm,	Y =  133.000  mm,	Z =   15.000 mm,
	W =-180.000 deg,	P =   0.000 deg,	R =    90.000 deg
};
P[6679]{
   GP1:
	UF : 1, UT : 4,		CONFIG : 'N U T, 0, 0, 0',
	X =  109.000  mm,	Y =  133.000  mm,	Z =   15.000 mm,
	W =-180.000 deg,	P =   0.000 deg,	R =    90.000 deg
};
P[6680]{
   GP1:
	UF : 1, UT : 4,		CONFIG : 'N U T, 0, 0, 0',
	X =  109.000  mm,	Y =  133.000  mm,	Z =   -1.000 mm,
	W =-180.000 deg,	P =   0.000 deg,	R =    90.000 deg
};
P[6681]{
   GP1:
	UF : 1, UT : 4,		CONFIG : 'N U T, 0, 0, 0',
	X =  109.000  mm,	Y =  133.000  mm,	Z =   15.000 mm,
	W =-180.000 deg,	P =   0.000 deg,	R =    90.000 deg
};
P[6718]{
   GP1:
	UF : 1, UT : 4,		CONFIG : 'N U T, 0, 0, 0',
	X =  148.000  mm,	Y =  133.000  mm,	Z =   15.000 mm,
	W =-180.000 deg,	P =   0.000 deg,	R =    90.000 deg
};
P[6719]{
   GP1:
	UF : 1, UT : 4,		CONFIG : 'N U T, 0, 0, 0',
	X =  148.000  mm,	Y =  133.000  mm,	Z =   -1.000 mm,
	W =-180.000 deg,	P =   0.000 deg,	R =    90.000 deg
};
P[6720]{
   GP1:
	UF : 1, UT : 4,		CONFIG : 'N U T, 0, 0, 0',
	X =  148.000  mm,	Y =  133.000  mm,	Z =   15.000 mm,
	W =-180.000 deg,	P =   0.000 deg,	R =    90.000 deg
};
P[6721]{
   GP1:
	UF : 1, UT : 4,		CONFIG : 'N U T, 0, 0, 0',
	X =  151.000  mm,	Y =  133.000  mm,	Z =   15.000 mm,
	W =-180.000 deg,	P =   0.000 deg,	R =    90.000 deg
};
P[6722]{
   GP1:
	UF : 1, UT : 4,		CONFIG : 'N U T, 0, 0, 0',
	X =  151.000  mm,	Y =  133.000  mm,	Z =   -1.000 mm,
	W =-180.000 deg,	P =   0.000 deg,	R =    90.000 deg
};
P[6723]{
   GP1:
	UF : 1, UT : 4,		CONFIG : 'N U T, 0, 0, 0',
	X =  151.000  mm,	Y =  133.000  mm,	Z =   15.000 mm,
	W =-180.000 deg,	P =   0.000 deg,	R =    90.000 deg
};
P[6730]{
   GP1:
	UF : 1, UT : 4,		CONFIG : 'N U T, 0, 0, 0',
	X =  19.000  mm,	Y =  136.000  mm,	Z =   15.000 mm,
	W =-180.000 deg,	P =   0.000 deg,	R =    90.000 deg
};
P[6731]{
   GP1:
	UF : 1, UT : 4,		CONFIG : 'N U T, 0, 0, 0',
	X =  19.000  mm,	Y =  136.000  mm,	Z =   -1.000 mm,
	W =-180.000 deg,	P =   0.000 deg,	R =    90.000 deg
};
P[6732]{
   GP1:
	UF : 1, UT : 4,		CONFIG : 'N U T, 0, 0, 0',
	X =  19.000  mm,	Y =  136.000  mm,	Z =   15.000 mm,
	W =-180.000 deg,	P =   0.000 deg,	R =    90.000 deg
};
P[6733]{
   GP1:
	UF : 1, UT : 4,		CONFIG : 'N U T, 0, 0, 0',
	X =  22.000  mm,	Y =  136.000  mm,	Z =   15.000 mm,
	W =-180.000 deg,	P =   0.000 deg,	R =    90.000 deg
};
P[6734]{
   GP1:
	UF : 1, UT : 4,		CONFIG : 'N U T, 0, 0, 0',
	X =  22.000  mm,	Y =  136.000  mm,	Z =   -1.000 mm,
	W =-180.000 deg,	P =   0.000 deg,	R =    90.000 deg
};
P[6735]{
   GP1:
	UF : 1, UT : 4,		CONFIG : 'N U T, 0, 0, 0',
	X =  22.000  mm,	Y =  136.000  mm,	Z =   15.000 mm,
	W =-180.000 deg,	P =   0.000 deg,	R =    90.000 deg
};
P[6748]{
   GP1:
	UF : 1, UT : 4,		CONFIG : 'N U T, 0, 0, 0',
	X =  37.000  mm,	Y =  136.000  mm,	Z =   15.000 mm,
	W =-180.000 deg,	P =   0.000 deg,	R =    90.000 deg
};
P[6749]{
   GP1:
	UF : 1, UT : 4,		CONFIG : 'N U T, 0, 0, 0',
	X =  37.000  mm,	Y =  136.000  mm,	Z =   -1.000 mm,
	W =-180.000 deg,	P =   0.000 deg,	R =    90.000 deg
};
P[6750]{
   GP1:
	UF : 1, UT : 4,		CONFIG : 'N U T, 0, 0, 0',
	X =  37.000  mm,	Y =  136.000  mm,	Z =   15.000 mm,
	W =-180.000 deg,	P =   0.000 deg,	R =    90.000 deg
};
P[6751]{
   GP1:
	UF : 1, UT : 4,		CONFIG : 'N U T, 0, 0, 0',
	X =  40.000  mm,	Y =  136.000  mm,	Z =   15.000 mm,
	W =-180.000 deg,	P =   0.000 deg,	R =    90.000 deg
};
P[6752]{
   GP1:
	UF : 1, UT : 4,		CONFIG : 'N U T, 0, 0, 0',
	X =  40.000  mm,	Y =  136.000  mm,	Z =   -1.000 mm,
	W =-180.000 deg,	P =   0.000 deg,	R =    90.000 deg
};
P[6753]{
   GP1:
	UF : 1, UT : 4,		CONFIG : 'N U T, 0, 0, 0',
	X =  40.000  mm,	Y =  136.000  mm,	Z =   15.000 mm,
	W =-180.000 deg,	P =   0.000 deg,	R =    90.000 deg
};
P[6754]{
   GP1:
	UF : 1, UT : 4,		CONFIG : 'N U T, 0, 0, 0',
	X =  43.000  mm,	Y =  136.000  mm,	Z =   15.000 mm,
	W =-180.000 deg,	P =   0.000 deg,	R =    90.000 deg
};
P[6755]{
   GP1:
	UF : 1, UT : 4,		CONFIG : 'N U T, 0, 0, 0',
	X =  43.000  mm,	Y =  136.000  mm,	Z =   -1.000 mm,
	W =-180.000 deg,	P =   0.000 deg,	R =    90.000 deg
};
P[6756]{
   GP1:
	UF : 1, UT : 4,		CONFIG : 'N U T, 0, 0, 0',
	X =  43.000  mm,	Y =  136.000  mm,	Z =   15.000 mm,
	W =-180.000 deg,	P =   0.000 deg,	R =    90.000 deg
};
P[6772]{
   GP1:
	UF : 1, UT : 4,		CONFIG : 'N U T, 0, 0, 0',
	X =  61.000  mm,	Y =  136.000  mm,	Z =   15.000 mm,
	W =-180.000 deg,	P =   0.000 deg,	R =    90.000 deg
};
P[6773]{
   GP1:
	UF : 1, UT : 4,		CONFIG : 'N U T, 0, 0, 0',
	X =  61.000  mm,	Y =  136.000  mm,	Z =   -1.000 mm,
	W =-180.000 deg,	P =   0.000 deg,	R =    90.000 deg
};
P[6774]{
   GP1:
	UF : 1, UT : 4,		CONFIG : 'N U T, 0, 0, 0',
	X =  61.000  mm,	Y =  136.000  mm,	Z =   15.000 mm,
	W =-180.000 deg,	P =   0.000 deg,	R =    90.000 deg
};
P[6781]{
   GP1:
	UF : 1, UT : 4,		CONFIG : 'N U T, 0, 0, 0',
	X =  109.000  mm,	Y =  136.000  mm,	Z =   15.000 mm,
	W =-180.000 deg,	P =   0.000 deg,	R =    90.000 deg
};
P[6782]{
   GP1:
	UF : 1, UT : 4,		CONFIG : 'N U T, 0, 0, 0',
	X =  109.000  mm,	Y =  136.000  mm,	Z =   -1.000 mm,
	W =-180.000 deg,	P =   0.000 deg,	R =    90.000 deg
};
P[6783]{
   GP1:
	UF : 1, UT : 4,		CONFIG : 'N U T, 0, 0, 0',
	X =  109.000  mm,	Y =  136.000  mm,	Z =   15.000 mm,
	W =-180.000 deg,	P =   0.000 deg,	R =    90.000 deg
};
P[6820]{
   GP1:
	UF : 1, UT : 4,		CONFIG : 'N U T, 0, 0, 0',
	X =  148.000  mm,	Y =  136.000  mm,	Z =   15.000 mm,
	W =-180.000 deg,	P =   0.000 deg,	R =    90.000 deg
};
P[6821]{
   GP1:
	UF : 1, UT : 4,		CONFIG : 'N U T, 0, 0, 0',
	X =  148.000  mm,	Y =  136.000  mm,	Z =   -1.000 mm,
	W =-180.000 deg,	P =   0.000 deg,	R =    90.000 deg
};
P[6822]{
   GP1:
	UF : 1, UT : 4,		CONFIG : 'N U T, 0, 0, 0',
	X =  148.000  mm,	Y =  136.000  mm,	Z =   15.000 mm,
	W =-180.000 deg,	P =   0.000 deg,	R =    90.000 deg
};
P[6823]{
   GP1:
	UF : 1, UT : 4,		CONFIG : 'N U T, 0, 0, 0',
	X =  151.000  mm,	Y =  136.000  mm,	Z =   15.000 mm,
	W =-180.000 deg,	P =   0.000 deg,	R =    90.000 deg
};
P[6824]{
   GP1:
	UF : 1, UT : 4,		CONFIG : 'N U T, 0, 0, 0',
	X =  151.000  mm,	Y =  136.000  mm,	Z =   -1.000 mm,
	W =-180.000 deg,	P =   0.000 deg,	R =    90.000 deg
};
P[6825]{
   GP1:
	UF : 1, UT : 4,		CONFIG : 'N U T, 0, 0, 0',
	X =  151.000  mm,	Y =  136.000  mm,	Z =   15.000 mm,
	W =-180.000 deg,	P =   0.000 deg,	R =    90.000 deg
};
P[6832]{
   GP1:
	UF : 1, UT : 4,		CONFIG : 'N U T, 0, 0, 0',
	X =  19.000  mm,	Y =  139.000  mm,	Z =   15.000 mm,
	W =-180.000 deg,	P =   0.000 deg,	R =    90.000 deg
};
P[6833]{
   GP1:
	UF : 1, UT : 4,		CONFIG : 'N U T, 0, 0, 0',
	X =  19.000  mm,	Y =  139.000  mm,	Z =   -1.000 mm,
	W =-180.000 deg,	P =   0.000 deg,	R =    90.000 deg
};
P[6834]{
   GP1:
	UF : 1, UT : 4,		CONFIG : 'N U T, 0, 0, 0',
	X =  19.000  mm,	Y =  139.000  mm,	Z =   15.000 mm,
	W =-180.000 deg,	P =   0.000 deg,	R =    90.000 deg
};
P[6850]{
   GP1:
	UF : 1, UT : 4,		CONFIG : 'N U T, 0, 0, 0',
	X =  37.000  mm,	Y =  139.000  mm,	Z =   15.000 mm,
	W =-180.000 deg,	P =   0.000 deg,	R =    90.000 deg
};
P[6851]{
   GP1:
	UF : 1, UT : 4,		CONFIG : 'N U T, 0, 0, 0',
	X =  37.000  mm,	Y =  139.000  mm,	Z =   -1.000 mm,
	W =-180.000 deg,	P =   0.000 deg,	R =    90.000 deg
};
P[6852]{
   GP1:
	UF : 1, UT : 4,		CONFIG : 'N U T, 0, 0, 0',
	X =  37.000  mm,	Y =  139.000  mm,	Z =   15.000 mm,
	W =-180.000 deg,	P =   0.000 deg,	R =    90.000 deg
};
P[6853]{
   GP1:
	UF : 1, UT : 4,		CONFIG : 'N U T, 0, 0, 0',
	X =  40.000  mm,	Y =  139.000  mm,	Z =   15.000 mm,
	W =-180.000 deg,	P =   0.000 deg,	R =    90.000 deg
};
P[6854]{
   GP1:
	UF : 1, UT : 4,		CONFIG : 'N U T, 0, 0, 0',
	X =  40.000  mm,	Y =  139.000  mm,	Z =   -1.000 mm,
	W =-180.000 deg,	P =   0.000 deg,	R =    90.000 deg
};
P[6855]{
   GP1:
	UF : 1, UT : 4,		CONFIG : 'N U T, 0, 0, 0',
	X =  40.000  mm,	Y =  139.000  mm,	Z =   15.000 mm,
	W =-180.000 deg,	P =   0.000 deg,	R =    90.000 deg
};
P[6886]{
   GP1:
	UF : 1, UT : 4,		CONFIG : 'N U T, 0, 0, 0',
	X =  109.000  mm,	Y =  139.000  mm,	Z =   15.000 mm,
	W =-180.000 deg,	P =   0.000 deg,	R =    90.000 deg
};
P[6887]{
   GP1:
	UF : 1, UT : 4,		CONFIG : 'N U T, 0, 0, 0',
	X =  109.000  mm,	Y =  139.000  mm,	Z =   -1.000 mm,
	W =-180.000 deg,	P =   0.000 deg,	R =    90.000 deg
};
P[6888]{
   GP1:
	UF : 1, UT : 4,		CONFIG : 'N U T, 0, 0, 0',
	X =  109.000  mm,	Y =  139.000  mm,	Z =   15.000 mm,
	W =-180.000 deg,	P =   0.000 deg,	R =    90.000 deg
};
P[6889]{
   GP1:
	UF : 1, UT : 4,		CONFIG : 'N U T, 0, 0, 0',
	X =  112.000  mm,	Y =  139.000  mm,	Z =   15.000 mm,
	W =-180.000 deg,	P =   0.000 deg,	R =    90.000 deg
};
P[6890]{
   GP1:
	UF : 1, UT : 4,		CONFIG : 'N U T, 0, 0, 0',
	X =  112.000  mm,	Y =  139.000  mm,	Z =   -1.000 mm,
	W =-180.000 deg,	P =   0.000 deg,	R =    90.000 deg
};
P[6891]{
   GP1:
	UF : 1, UT : 4,		CONFIG : 'N U T, 0, 0, 0',
	X =  112.000  mm,	Y =  139.000  mm,	Z =   15.000 mm,
	W =-180.000 deg,	P =   0.000 deg,	R =    90.000 deg
};
P[6904]{
   GP1:
	UF : 1, UT : 4,		CONFIG : 'N U T, 0, 0, 0',
	X =  127.000  mm,	Y =  139.000  mm,	Z =   15.000 mm,
	W =-180.000 deg,	P =   0.000 deg,	R =    90.000 deg
};
P[6905]{
   GP1:
	UF : 1, UT : 4,		CONFIG : 'N U T, 0, 0, 0',
	X =  127.000  mm,	Y =  139.000  mm,	Z =   -1.000 mm,
	W =-180.000 deg,	P =   0.000 deg,	R =    90.000 deg
};
P[6906]{
   GP1:
	UF : 1, UT : 4,		CONFIG : 'N U T, 0, 0, 0',
	X =  127.000  mm,	Y =  139.000  mm,	Z =   15.000 mm,
	W =-180.000 deg,	P =   0.000 deg,	R =    90.000 deg
};
P[6907]{
   GP1:
	UF : 1, UT : 4,		CONFIG : 'N U T, 0, 0, 0',
	X =  130.000  mm,	Y =  139.000  mm,	Z =   15.000 mm,
	W =-180.000 deg,	P =   0.000 deg,	R =    90.000 deg
};
P[6908]{
   GP1:
	UF : 1, UT : 4,		CONFIG : 'N U T, 0, 0, 0',
	X =  130.000  mm,	Y =  139.000  mm,	Z =   -1.000 mm,
	W =-180.000 deg,	P =   0.000 deg,	R =    90.000 deg
};
P[6909]{
   GP1:
	UF : 1, UT : 4,		CONFIG : 'N U T, 0, 0, 0',
	X =  130.000  mm,	Y =  139.000  mm,	Z =   15.000 mm,
	W =-180.000 deg,	P =   0.000 deg,	R =    90.000 deg
};
P[6910]{
   GP1:
	UF : 1, UT : 4,		CONFIG : 'N U T, 0, 0, 0',
	X =  133.000  mm,	Y =  139.000  mm,	Z =   15.000 mm,
	W =-180.000 deg,	P =   0.000 deg,	R =    90.000 deg
};
P[6911]{
   GP1:
	UF : 1, UT : 4,		CONFIG : 'N U T, 0, 0, 0',
	X =  133.000  mm,	Y =  139.000  mm,	Z =   -1.000 mm,
	W =-180.000 deg,	P =   0.000 deg,	R =    90.000 deg
};
P[6912]{
   GP1:
	UF : 1, UT : 4,		CONFIG : 'N U T, 0, 0, 0',
	X =  133.000  mm,	Y =  139.000  mm,	Z =   15.000 mm,
	W =-180.000 deg,	P =   0.000 deg,	R =    90.000 deg
};
P[6922]{
   GP1:
	UF : 1, UT : 4,		CONFIG : 'N U T, 0, 0, 0',
	X =  145.000  mm,	Y =  139.000  mm,	Z =   15.000 mm,
	W =-180.000 deg,	P =   0.000 deg,	R =    90.000 deg
};
P[6923]{
   GP1:
	UF : 1, UT : 4,		CONFIG : 'N U T, 0, 0, 0',
	X =  145.000  mm,	Y =  139.000  mm,	Z =   -1.000 mm,
	W =-180.000 deg,	P =   0.000 deg,	R =    90.000 deg
};
P[6924]{
   GP1:
	UF : 1, UT : 4,		CONFIG : 'N U T, 0, 0, 0',
	X =  145.000  mm,	Y =  139.000  mm,	Z =   15.000 mm,
	W =-180.000 deg,	P =   0.000 deg,	R =    90.000 deg
};
P[6925]{
   GP1:
	UF : 1, UT : 4,		CONFIG : 'N U T, 0, 0, 0',
	X =  148.000  mm,	Y =  139.000  mm,	Z =   15.000 mm,
	W =-180.000 deg,	P =   0.000 deg,	R =    90.000 deg
};
P[6926]{
   GP1:
	UF : 1, UT : 4,		CONFIG : 'N U T, 0, 0, 0',
	X =  148.000  mm,	Y =  139.000  mm,	Z =   -1.000 mm,
	W =-180.000 deg,	P =   0.000 deg,	R =    90.000 deg
};
P[6927]{
   GP1:
	UF : 1, UT : 4,		CONFIG : 'N U T, 0, 0, 0',
	X =  148.000  mm,	Y =  139.000  mm,	Z =   15.000 mm,
	W =-180.000 deg,	P =   0.000 deg,	R =    90.000 deg
};
P[6928]{
   GP1:
	UF : 1, UT : 4,		CONFIG : 'N U T, 0, 0, 0',
	X =  151.000  mm,	Y =  139.000  mm,	Z =   15.000 mm,
	W =-180.000 deg,	P =   0.000 deg,	R =    90.000 deg
};
P[6929]{
   GP1:
	UF : 1, UT : 4,		CONFIG : 'N U T, 0, 0, 0',
	X =  151.000  mm,	Y =  139.000  mm,	Z =   -1.000 mm,
	W =-180.000 deg,	P =   0.000 deg,	R =    90.000 deg
};
P[6930]{
   GP1:
	UF : 1, UT : 4,		CONFIG : 'N U T, 0, 0, 0',
	X =  151.000  mm,	Y =  139.000  mm,	Z =   15.000 mm,
	W =-180.000 deg,	P =   0.000 deg,	R =    90.000 deg
};
P[6934]{
   GP1:
	UF : 1, UT : 4,		CONFIG : 'N U T, 0, 0, 0',
	X =  19.000  mm,	Y =  142.000  mm,	Z =   15.000 mm,
	W =-180.000 deg,	P =   0.000 deg,	R =    90.000 deg
};
P[6935]{
   GP1:
	UF : 1, UT : 4,		CONFIG : 'N U T, 0, 0, 0',
	X =  19.000  mm,	Y =  142.000  mm,	Z =   -1.000 mm,
	W =-180.000 deg,	P =   0.000 deg,	R =    90.000 deg
};
P[6936]{
   GP1:
	UF : 1, UT : 4,		CONFIG : 'N U T, 0, 0, 0',
	X =  19.000  mm,	Y =  142.000  mm,	Z =   15.000 mm,
	W =-180.000 deg,	P =   0.000 deg,	R =    90.000 deg
};
P[6973]{
   GP1:
	UF : 1, UT : 4,		CONFIG : 'N U T, 0, 0, 0',
	X =  58.000  mm,	Y =  142.000  mm,	Z =   15.000 mm,
	W =-180.000 deg,	P =   0.000 deg,	R =    90.000 deg
};
P[6974]{
   GP1:
	UF : 1, UT : 4,		CONFIG : 'N U T, 0, 0, 0',
	X =  58.000  mm,	Y =  142.000  mm,	Z =   -1.000 mm,
	W =-180.000 deg,	P =   0.000 deg,	R =    90.000 deg
};
P[6975]{
   GP1:
	UF : 1, UT : 4,		CONFIG : 'N U T, 0, 0, 0',
	X =  58.000  mm,	Y =  142.000  mm,	Z =   15.000 mm,
	W =-180.000 deg,	P =   0.000 deg,	R =    90.000 deg
};
P[6976]{
   GP1:
	UF : 1, UT : 4,		CONFIG : 'N U T, 0, 0, 0',
	X =  61.000  mm,	Y =  142.000  mm,	Z =   15.000 mm,
	W =-180.000 deg,	P =   0.000 deg,	R =    90.000 deg
};
P[6977]{
   GP1:
	UF : 1, UT : 4,		CONFIG : 'N U T, 0, 0, 0',
	X =  61.000  mm,	Y =  142.000  mm,	Z =   -1.000 mm,
	W =-180.000 deg,	P =   0.000 deg,	R =    90.000 deg
};
P[6978]{
   GP1:
	UF : 1, UT : 4,		CONFIG : 'N U T, 0, 0, 0',
	X =  61.000  mm,	Y =  142.000  mm,	Z =   15.000 mm,
	W =-180.000 deg,	P =   0.000 deg,	R =    90.000 deg
};
P[7003]{
   GP1:
	UF : 1, UT : 4,		CONFIG : 'N U T, 0, 0, 0',
	X =  109.000  mm,	Y =  142.000  mm,	Z =   15.000 mm,
	W =-180.000 deg,	P =   0.000 deg,	R =    90.000 deg
};
P[7004]{
   GP1:
	UF : 1, UT : 4,		CONFIG : 'N U T, 0, 0, 0',
	X =  109.000  mm,	Y =  142.000  mm,	Z =   -1.000 mm,
	W =-180.000 deg,	P =   0.000 deg,	R =    90.000 deg
};
P[7005]{
   GP1:
	UF : 1, UT : 4,		CONFIG : 'N U T, 0, 0, 0',
	X =  109.000  mm,	Y =  142.000  mm,	Z =   15.000 mm,
	W =-180.000 deg,	P =   0.000 deg,	R =    90.000 deg
};
P[7006]{
   GP1:
	UF : 1, UT : 4,		CONFIG : 'N U T, 0, 0, 0',
	X =  112.000  mm,	Y =  142.000  mm,	Z =   15.000 mm,
	W =-180.000 deg,	P =   0.000 deg,	R =    90.000 deg
};
P[7007]{
   GP1:
	UF : 1, UT : 4,		CONFIG : 'N U T, 0, 0, 0',
	X =  112.000  mm,	Y =  142.000  mm,	Z =   -1.000 mm,
	W =-180.000 deg,	P =   0.000 deg,	R =    90.000 deg
};
P[7008]{
   GP1:
	UF : 1, UT : 4,		CONFIG : 'N U T, 0, 0, 0',
	X =  112.000  mm,	Y =  142.000  mm,	Z =   15.000 mm,
	W =-180.000 deg,	P =   0.000 deg,	R =    90.000 deg
};
P[7015]{
   GP1:
	UF : 1, UT : 4,		CONFIG : 'N U T, 0, 0, 0',
	X =  121.000  mm,	Y =  142.000  mm,	Z =   15.000 mm,
	W =-180.000 deg,	P =   0.000 deg,	R =    90.000 deg
};
P[7016]{
   GP1:
	UF : 1, UT : 4,		CONFIG : 'N U T, 0, 0, 0',
	X =  121.000  mm,	Y =  142.000  mm,	Z =   -1.000 mm,
	W =-180.000 deg,	P =   0.000 deg,	R =    90.000 deg
};
P[7017]{
   GP1:
	UF : 1, UT : 4,		CONFIG : 'N U T, 0, 0, 0',
	X =  121.000  mm,	Y =  142.000  mm,	Z =   15.000 mm,
	W =-180.000 deg,	P =   0.000 deg,	R =    90.000 deg
};
P[7018]{
   GP1:
	UF : 1, UT : 4,		CONFIG : 'N U T, 0, 0, 0',
	X =  124.000  mm,	Y =  142.000  mm,	Z =   15.000 mm,
	W =-180.000 deg,	P =   0.000 deg,	R =    90.000 deg
};
P[7019]{
   GP1:
	UF : 1, UT : 4,		CONFIG : 'N U T, 0, 0, 0',
	X =  124.000  mm,	Y =  142.000  mm,	Z =   -1.000 mm,
	W =-180.000 deg,	P =   0.000 deg,	R =    90.000 deg
};
P[7020]{
   GP1:
	UF : 1, UT : 4,		CONFIG : 'N U T, 0, 0, 0',
	X =  124.000  mm,	Y =  142.000  mm,	Z =   15.000 mm,
	W =-180.000 deg,	P =   0.000 deg,	R =    90.000 deg
};
P[7021]{
   GP1:
	UF : 1, UT : 4,		CONFIG : 'N U T, 0, 0, 0',
	X =  127.000  mm,	Y =  142.000  mm,	Z =   15.000 mm,
	W =-180.000 deg,	P =   0.000 deg,	R =    90.000 deg
};
P[7022]{
   GP1:
	UF : 1, UT : 4,		CONFIG : 'N U T, 0, 0, 0',
	X =  127.000  mm,	Y =  142.000  mm,	Z =   -1.000 mm,
	W =-180.000 deg,	P =   0.000 deg,	R =    90.000 deg
};
P[7023]{
   GP1:
	UF : 1, UT : 4,		CONFIG : 'N U T, 0, 0, 0',
	X =  127.000  mm,	Y =  142.000  mm,	Z =   15.000 mm,
	W =-180.000 deg,	P =   0.000 deg,	R =    90.000 deg
};
P[7024]{
   GP1:
	UF : 1, UT : 4,		CONFIG : 'N U T, 0, 0, 0',
	X =  130.000  mm,	Y =  142.000  mm,	Z =   15.000 mm,
	W =-180.000 deg,	P =   0.000 deg,	R =    90.000 deg
};
P[7025]{
   GP1:
	UF : 1, UT : 4,		CONFIG : 'N U T, 0, 0, 0',
	X =  130.000  mm,	Y =  142.000  mm,	Z =   -1.000 mm,
	W =-180.000 deg,	P =   0.000 deg,	R =    90.000 deg
};
P[7026]{
   GP1:
	UF : 1, UT : 4,		CONFIG : 'N U T, 0, 0, 0',
	X =  130.000  mm,	Y =  142.000  mm,	Z =   15.000 mm,
	W =-180.000 deg,	P =   0.000 deg,	R =    90.000 deg
};
P[7033]{
   GP1:
	UF : 1, UT : 4,		CONFIG : 'N U T, 0, 0, 0',
	X =  139.000  mm,	Y =  142.000  mm,	Z =   15.000 mm,
	W =-180.000 deg,	P =   0.000 deg,	R =    90.000 deg
};
P[7034]{
   GP1:
	UF : 1, UT : 4,		CONFIG : 'N U T, 0, 0, 0',
	X =  139.000  mm,	Y =  142.000  mm,	Z =   -1.000 mm,
	W =-180.000 deg,	P =   0.000 deg,	R =    90.000 deg
};
P[7035]{
   GP1:
	UF : 1, UT : 4,		CONFIG : 'N U T, 0, 0, 0',
	X =  139.000  mm,	Y =  142.000  mm,	Z =   15.000 mm,
	W =-180.000 deg,	P =   0.000 deg,	R =    90.000 deg
};
P[7036]{
   GP1:
	UF : 1, UT : 4,		CONFIG : 'N U T, 0, 0, 0',
	X =  142.000  mm,	Y =  142.000  mm,	Z =   15.000 mm,
	W =-180.000 deg,	P =   0.000 deg,	R =    90.000 deg
};
P[7037]{
   GP1:
	UF : 1, UT : 4,		CONFIG : 'N U T, 0, 0, 0',
	X =  142.000  mm,	Y =  142.000  mm,	Z =   -1.000 mm,
	W =-180.000 deg,	P =   0.000 deg,	R =    90.000 deg
};
P[7038]{
   GP1:
	UF : 1, UT : 4,		CONFIG : 'N U T, 0, 0, 0',
	X =  142.000  mm,	Y =  142.000  mm,	Z =   15.000 mm,
	W =-180.000 deg,	P =   0.000 deg,	R =    90.000 deg
};
P[7039]{
   GP1:
	UF : 1, UT : 4,		CONFIG : 'N U T, 0, 0, 0',
	X =  145.000  mm,	Y =  142.000  mm,	Z =   15.000 mm,
	W =-180.000 deg,	P =   0.000 deg,	R =    90.000 deg
};
P[7040]{
   GP1:
	UF : 1, UT : 4,		CONFIG : 'N U T, 0, 0, 0',
	X =  145.000  mm,	Y =  142.000  mm,	Z =   -1.000 mm,
	W =-180.000 deg,	P =   0.000 deg,	R =    90.000 deg
};
P[7041]{
   GP1:
	UF : 1, UT : 4,		CONFIG : 'N U T, 0, 0, 0',
	X =  145.000  mm,	Y =  142.000  mm,	Z =   15.000 mm,
	W =-180.000 deg,	P =   0.000 deg,	R =    90.000 deg
};
P[7042]{
   GP1:
	UF : 1, UT : 4,		CONFIG : 'N U T, 0, 0, 0',
	X =  148.000  mm,	Y =  142.000  mm,	Z =   15.000 mm,
	W =-180.000 deg,	P =   0.000 deg,	R =    90.000 deg
};
P[7043]{
   GP1:
	UF : 1, UT : 4,		CONFIG : 'N U T, 0, 0, 0',
	X =  148.000  mm,	Y =  142.000  mm,	Z =   -1.000 mm,
	W =-180.000 deg,	P =   0.000 deg,	R =    90.000 deg
};
P[7044]{
   GP1:
	UF : 1, UT : 4,		CONFIG : 'N U T, 0, 0, 0',
	X =  148.000  mm,	Y =  142.000  mm,	Z =   15.000 mm,
	W =-180.000 deg,	P =   0.000 deg,	R =    90.000 deg
};
P[7045]{
   GP1:
	UF : 1, UT : 4,		CONFIG : 'N U T, 0, 0, 0',
	X =  151.000  mm,	Y =  142.000  mm,	Z =   15.000 mm,
	W =-180.000 deg,	P =   0.000 deg,	R =    90.000 deg
};
P[7046]{
   GP1:
	UF : 1, UT : 4,		CONFIG : 'N U T, 0, 0, 0',
	X =  151.000  mm,	Y =  142.000  mm,	Z =   -1.000 mm,
	W =-180.000 deg,	P =   0.000 deg,	R =    90.000 deg
};
P[7047]{
   GP1:
	UF : 1, UT : 4,		CONFIG : 'N U T, 0, 0, 0',
	X =  151.000  mm,	Y =  142.000  mm,	Z =   15.000 mm,
	W =-180.000 deg,	P =   0.000 deg,	R =    90.000 deg
};
P[7051]{
   GP1:
	UF : 1, UT : 4,		CONFIG : 'N U T, 0, 0, 0',
	X =  19.000  mm,	Y =  145.000  mm,	Z =   15.000 mm,
	W =-180.000 deg,	P =   0.000 deg,	R =    90.000 deg
};
P[7052]{
   GP1:
	UF : 1, UT : 4,		CONFIG : 'N U T, 0, 0, 0',
	X =  19.000  mm,	Y =  145.000  mm,	Z =   -1.000 mm,
	W =-180.000 deg,	P =   0.000 deg,	R =    90.000 deg
};
P[7053]{
   GP1:
	UF : 1, UT : 4,		CONFIG : 'N U T, 0, 0, 0',
	X =  19.000  mm,	Y =  145.000  mm,	Z =   15.000 mm,
	W =-180.000 deg,	P =   0.000 deg,	R =    90.000 deg
};
P[7069]{
   GP1:
	UF : 1, UT : 4,		CONFIG : 'N U T, 0, 0, 0',
	X =  37.000  mm,	Y =  145.000  mm,	Z =   15.000 mm,
	W =-180.000 deg,	P =   0.000 deg,	R =    90.000 deg
};
P[7070]{
   GP1:
	UF : 1, UT : 4,		CONFIG : 'N U T, 0, 0, 0',
	X =  37.000  mm,	Y =  145.000  mm,	Z =   -1.000 mm,
	W =-180.000 deg,	P =   0.000 deg,	R =    90.000 deg
};
P[7071]{
   GP1:
	UF : 1, UT : 4,		CONFIG : 'N U T, 0, 0, 0',
	X =  37.000  mm,	Y =  145.000  mm,	Z =   15.000 mm,
	W =-180.000 deg,	P =   0.000 deg,	R =    90.000 deg
};
P[7072]{
   GP1:
	UF : 1, UT : 4,		CONFIG : 'N U T, 0, 0, 0',
	X =  40.000  mm,	Y =  145.000  mm,	Z =   15.000 mm,
	W =-180.000 deg,	P =   0.000 deg,	R =    90.000 deg
};
P[7073]{
   GP1:
	UF : 1, UT : 4,		CONFIG : 'N U T, 0, 0, 0',
	X =  40.000  mm,	Y =  145.000  mm,	Z =   -1.000 mm,
	W =-180.000 deg,	P =   0.000 deg,	R =    90.000 deg
};
P[7074]{
   GP1:
	UF : 1, UT : 4,		CONFIG : 'N U T, 0, 0, 0',
	X =  40.000  mm,	Y =  145.000  mm,	Z =   15.000 mm,
	W =-180.000 deg,	P =   0.000 deg,	R =    90.000 deg
};
P[7075]{
   GP1:
	UF : 1, UT : 4,		CONFIG : 'N U T, 0, 0, 0',
	X =  43.000  mm,	Y =  145.000  mm,	Z =   15.000 mm,
	W =-180.000 deg,	P =   0.000 deg,	R =    90.000 deg
};
P[7076]{
   GP1:
	UF : 1, UT : 4,		CONFIG : 'N U T, 0, 0, 0',
	X =  43.000  mm,	Y =  145.000  mm,	Z =   -1.000 mm,
	W =-180.000 deg,	P =   0.000 deg,	R =    90.000 deg
};
P[7077]{
   GP1:
	UF : 1, UT : 4,		CONFIG : 'N U T, 0, 0, 0',
	X =  43.000  mm,	Y =  145.000  mm,	Z =   15.000 mm,
	W =-180.000 deg,	P =   0.000 deg,	R =    90.000 deg
};
P[7078]{
   GP1:
	UF : 1, UT : 4,		CONFIG : 'N U T, 0, 0, 0',
	X =  46.000  mm,	Y =  145.000  mm,	Z =   15.000 mm,
	W =-180.000 deg,	P =   0.000 deg,	R =    90.000 deg
};
P[7079]{
   GP1:
	UF : 1, UT : 4,		CONFIG : 'N U T, 0, 0, 0',
	X =  46.000  mm,	Y =  145.000  mm,	Z =   -1.000 mm,
	W =-180.000 deg,	P =   0.000 deg,	R =    90.000 deg
};
P[7080]{
   GP1:
	UF : 1, UT : 4,		CONFIG : 'N U T, 0, 0, 0',
	X =  46.000  mm,	Y =  145.000  mm,	Z =   15.000 mm,
	W =-180.000 deg,	P =   0.000 deg,	R =    90.000 deg
};
P[7081]{
   GP1:
	UF : 1, UT : 4,		CONFIG : 'N U T, 0, 0, 0',
	X =  49.000  mm,	Y =  145.000  mm,	Z =   15.000 mm,
	W =-180.000 deg,	P =   0.000 deg,	R =    90.000 deg
};
P[7082]{
   GP1:
	UF : 1, UT : 4,		CONFIG : 'N U T, 0, 0, 0',
	X =  49.000  mm,	Y =  145.000  mm,	Z =   -1.000 mm,
	W =-180.000 deg,	P =   0.000 deg,	R =    90.000 deg
};
P[7083]{
   GP1:
	UF : 1, UT : 4,		CONFIG : 'N U T, 0, 0, 0',
	X =  49.000  mm,	Y =  145.000  mm,	Z =   15.000 mm,
	W =-180.000 deg,	P =   0.000 deg,	R =    90.000 deg
};
P[7084]{
   GP1:
	UF : 1, UT : 4,		CONFIG : 'N U T, 0, 0, 0',
	X =  52.000  mm,	Y =  145.000  mm,	Z =   15.000 mm,
	W =-180.000 deg,	P =   0.000 deg,	R =    90.000 deg
};
P[7085]{
   GP1:
	UF : 1, UT : 4,		CONFIG : 'N U T, 0, 0, 0',
	X =  52.000  mm,	Y =  145.000  mm,	Z =   -1.000 mm,
	W =-180.000 deg,	P =   0.000 deg,	R =    90.000 deg
};
P[7086]{
   GP1:
	UF : 1, UT : 4,		CONFIG : 'N U T, 0, 0, 0',
	X =  52.000  mm,	Y =  145.000  mm,	Z =   15.000 mm,
	W =-180.000 deg,	P =   0.000 deg,	R =    90.000 deg
};
P[7087]{
   GP1:
	UF : 1, UT : 4,		CONFIG : 'N U T, 0, 0, 0',
	X =  55.000  mm,	Y =  145.000  mm,	Z =   15.000 mm,
	W =-180.000 deg,	P =   0.000 deg,	R =    90.000 deg
};
P[7088]{
   GP1:
	UF : 1, UT : 4,		CONFIG : 'N U T, 0, 0, 0',
	X =  55.000  mm,	Y =  145.000  mm,	Z =   -1.000 mm,
	W =-180.000 deg,	P =   0.000 deg,	R =    90.000 deg
};
P[7089]{
   GP1:
	UF : 1, UT : 4,		CONFIG : 'N U T, 0, 0, 0',
	X =  55.000  mm,	Y =  145.000  mm,	Z =   15.000 mm,
	W =-180.000 deg,	P =   0.000 deg,	R =    90.000 deg
};
P[7090]{
   GP1:
	UF : 1, UT : 4,		CONFIG : 'N U T, 0, 0, 0',
	X =  58.000  mm,	Y =  145.000  mm,	Z =   15.000 mm,
	W =-180.000 deg,	P =   0.000 deg,	R =    90.000 deg
};
P[7091]{
   GP1:
	UF : 1, UT : 4,		CONFIG : 'N U T, 0, 0, 0',
	X =  58.000  mm,	Y =  145.000  mm,	Z =   -1.000 mm,
	W =-180.000 deg,	P =   0.000 deg,	R =    90.000 deg
};
P[7092]{
   GP1:
	UF : 1, UT : 4,		CONFIG : 'N U T, 0, 0, 0',
	X =  58.000  mm,	Y =  145.000  mm,	Z =   15.000 mm,
	W =-180.000 deg,	P =   0.000 deg,	R =    90.000 deg
};
P[7093]{
   GP1:
	UF : 1, UT : 4,		CONFIG : 'N U T, 0, 0, 0',
	X =  61.000  mm,	Y =  145.000  mm,	Z =   15.000 mm,
	W =-180.000 deg,	P =   0.000 deg,	R =    90.000 deg
};
P[7094]{
   GP1:
	UF : 1, UT : 4,		CONFIG : 'N U T, 0, 0, 0',
	X =  61.000  mm,	Y =  145.000  mm,	Z =   -1.000 mm,
	W =-180.000 deg,	P =   0.000 deg,	R =    90.000 deg
};
P[7095]{
   GP1:
	UF : 1, UT : 4,		CONFIG : 'N U T, 0, 0, 0',
	X =  61.000  mm,	Y =  145.000  mm,	Z =   15.000 mm,
	W =-180.000 deg,	P =   0.000 deg,	R =    90.000 deg
};
P[7102]{
   GP1:
	UF : 1, UT : 4,		CONFIG : 'N U T, 0, 0, 0',
	X =  109.000  mm,	Y =  145.000  mm,	Z =   15.000 mm,
	W =-180.000 deg,	P =   0.000 deg,	R =    90.000 deg
};
P[7103]{
   GP1:
	UF : 1, UT : 4,		CONFIG : 'N U T, 0, 0, 0',
	X =  109.000  mm,	Y =  145.000  mm,	Z =   -1.000 mm,
	W =-180.000 deg,	P =   0.000 deg,	R =    90.000 deg
};
P[7104]{
   GP1:
	UF : 1, UT : 4,		CONFIG : 'N U T, 0, 0, 0',
	X =  109.000  mm,	Y =  145.000  mm,	Z =   15.000 mm,
	W =-180.000 deg,	P =   0.000 deg,	R =    90.000 deg
};
P[7117]{
   GP1:
	UF : 1, UT : 4,		CONFIG : 'N U T, 0, 0, 0',
	X =  124.000  mm,	Y =  145.000  mm,	Z =   15.000 mm,
	W =-180.000 deg,	P =   0.000 deg,	R =    90.000 deg
};
P[7118]{
   GP1:
	UF : 1, UT : 4,		CONFIG : 'N U T, 0, 0, 0',
	X =  124.000  mm,	Y =  145.000  mm,	Z =   -1.000 mm,
	W =-180.000 deg,	P =   0.000 deg,	R =    90.000 deg
};
P[7119]{
   GP1:
	UF : 1, UT : 4,		CONFIG : 'N U T, 0, 0, 0',
	X =  124.000  mm,	Y =  145.000  mm,	Z =   15.000 mm,
	W =-180.000 deg,	P =   0.000 deg,	R =    90.000 deg
};
P[7120]{
   GP1:
	UF : 1, UT : 4,		CONFIG : 'N U T, 0, 0, 0',
	X =  127.000  mm,	Y =  145.000  mm,	Z =   15.000 mm,
	W =-180.000 deg,	P =   0.000 deg,	R =    90.000 deg
};
P[7121]{
   GP1:
	UF : 1, UT : 4,		CONFIG : 'N U T, 0, 0, 0',
	X =  127.000  mm,	Y =  145.000  mm,	Z =   -1.000 mm,
	W =-180.000 deg,	P =   0.000 deg,	R =    90.000 deg
};
P[7122]{
   GP1:
	UF : 1, UT : 4,		CONFIG : 'N U T, 0, 0, 0',
	X =  127.000  mm,	Y =  145.000  mm,	Z =   15.000 mm,
	W =-180.000 deg,	P =   0.000 deg,	R =    90.000 deg
};
P[7123]{
   GP1:
	UF : 1, UT : 4,		CONFIG : 'N U T, 0, 0, 0',
	X =  130.000  mm,	Y =  145.000  mm,	Z =   15.000 mm,
	W =-180.000 deg,	P =   0.000 deg,	R =    90.000 deg
};
P[7124]{
   GP1:
	UF : 1, UT : 4,		CONFIG : 'N U T, 0, 0, 0',
	X =  130.000  mm,	Y =  145.000  mm,	Z =   -1.000 mm,
	W =-180.000 deg,	P =   0.000 deg,	R =    90.000 deg
};
P[7125]{
   GP1:
	UF : 1, UT : 4,		CONFIG : 'N U T, 0, 0, 0',
	X =  130.000  mm,	Y =  145.000  mm,	Z =   15.000 mm,
	W =-180.000 deg,	P =   0.000 deg,	R =    90.000 deg
};
P[7129]{
   GP1:
	UF : 1, UT : 4,		CONFIG : 'N U T, 0, 0, 0',
	X =  136.000  mm,	Y =  145.000  mm,	Z =   15.000 mm,
	W =-180.000 deg,	P =   0.000 deg,	R =    90.000 deg
};
P[7130]{
   GP1:
	UF : 1, UT : 4,		CONFIG : 'N U T, 0, 0, 0',
	X =  136.000  mm,	Y =  145.000  mm,	Z =   -1.000 mm,
	W =-180.000 deg,	P =   0.000 deg,	R =    90.000 deg
};
P[7131]{
   GP1:
	UF : 1, UT : 4,		CONFIG : 'N U T, 0, 0, 0',
	X =  136.000  mm,	Y =  145.000  mm,	Z =   15.000 mm,
	W =-180.000 deg,	P =   0.000 deg,	R =    90.000 deg
};
P[7132]{
   GP1:
	UF : 1, UT : 4,		CONFIG : 'N U T, 0, 0, 0',
	X =  139.000  mm,	Y =  145.000  mm,	Z =   15.000 mm,
	W =-180.000 deg,	P =   0.000 deg,	R =    90.000 deg
};
P[7133]{
   GP1:
	UF : 1, UT : 4,		CONFIG : 'N U T, 0, 0, 0',
	X =  139.000  mm,	Y =  145.000  mm,	Z =   -1.000 mm,
	W =-180.000 deg,	P =   0.000 deg,	R =    90.000 deg
};
P[7134]{
   GP1:
	UF : 1, UT : 4,		CONFIG : 'N U T, 0, 0, 0',
	X =  139.000  mm,	Y =  145.000  mm,	Z =   15.000 mm,
	W =-180.000 deg,	P =   0.000 deg,	R =    90.000 deg
};
P[7135]{
   GP1:
	UF : 1, UT : 4,		CONFIG : 'N U T, 0, 0, 0',
	X =  142.000  mm,	Y =  145.000  mm,	Z =   15.000 mm,
	W =-180.000 deg,	P =   0.000 deg,	R =    90.000 deg
};
P[7136]{
   GP1:
	UF : 1, UT : 4,		CONFIG : 'N U T, 0, 0, 0',
	X =  142.000  mm,	Y =  145.000  mm,	Z =   -1.000 mm,
	W =-180.000 deg,	P =   0.000 deg,	R =    90.000 deg
};
P[7137]{
   GP1:
	UF : 1, UT : 4,		CONFIG : 'N U T, 0, 0, 0',
	X =  142.000  mm,	Y =  145.000  mm,	Z =   15.000 mm,
	W =-180.000 deg,	P =   0.000 deg,	R =    90.000 deg
};
P[7138]{
   GP1:
	UF : 1, UT : 4,		CONFIG : 'N U T, 0, 0, 0',
	X =  145.000  mm,	Y =  145.000  mm,	Z =   15.000 mm,
	W =-180.000 deg,	P =   0.000 deg,	R =    90.000 deg
};
P[7139]{
   GP1:
	UF : 1, UT : 4,		CONFIG : 'N U T, 0, 0, 0',
	X =  145.000  mm,	Y =  145.000  mm,	Z =   -1.000 mm,
	W =-180.000 deg,	P =   0.000 deg,	R =    90.000 deg
};
P[7140]{
   GP1:
	UF : 1, UT : 4,		CONFIG : 'N U T, 0, 0, 0',
	X =  145.000  mm,	Y =  145.000  mm,	Z =   15.000 mm,
	W =-180.000 deg,	P =   0.000 deg,	R =    90.000 deg
};
P[7141]{
   GP1:
	UF : 1, UT : 4,		CONFIG : 'N U T, 0, 0, 0',
	X =  148.000  mm,	Y =  145.000  mm,	Z =   15.000 mm,
	W =-180.000 deg,	P =   0.000 deg,	R =    90.000 deg
};
P[7142]{
   GP1:
	UF : 1, UT : 4,		CONFIG : 'N U T, 0, 0, 0',
	X =  148.000  mm,	Y =  145.000  mm,	Z =   -1.000 mm,
	W =-180.000 deg,	P =   0.000 deg,	R =    90.000 deg
};
P[7143]{
   GP1:
	UF : 1, UT : 4,		CONFIG : 'N U T, 0, 0, 0',
	X =  148.000  mm,	Y =  145.000  mm,	Z =   15.000 mm,
	W =-180.000 deg,	P =   0.000 deg,	R =    90.000 deg
};
P[7144]{
   GP1:
	UF : 1, UT : 4,		CONFIG : 'N U T, 0, 0, 0',
	X =  151.000  mm,	Y =  145.000  mm,	Z =   15.000 mm,
	W =-180.000 deg,	P =   0.000 deg,	R =    90.000 deg
};
P[7145]{
   GP1:
	UF : 1, UT : 4,		CONFIG : 'N U T, 0, 0, 0',
	X =  151.000  mm,	Y =  145.000  mm,	Z =   -1.000 mm,
	W =-180.000 deg,	P =   0.000 deg,	R =    90.000 deg
};
P[7146]{
   GP1:
	UF : 1, UT : 4,		CONFIG : 'N U T, 0, 0, 0',
	X =  151.000  mm,	Y =  145.000  mm,	Z =   15.000 mm,
	W =-180.000 deg,	P =   0.000 deg,	R =    90.000 deg
};
P[7147]{
   GP1:
	UF : 1, UT : 4,		CONFIG : 'N U T, 0, 0, 0',
	X =  154.000  mm,	Y =  145.000  mm,	Z =   15.000 mm,
	W =-180.000 deg,	P =   0.000 deg,	R =    90.000 deg
};
P[7148]{
   GP1:
	UF : 1, UT : 4,		CONFIG : 'N U T, 0, 0, 0',
	X =  154.000  mm,	Y =  145.000  mm,	Z =   -1.000 mm,
	W =-180.000 deg,	P =   0.000 deg,	R =    90.000 deg
};
P[7149]{
   GP1:
	UF : 1, UT : 4,		CONFIG : 'N U T, 0, 0, 0',
	X =  154.000  mm,	Y =  145.000  mm,	Z =   15.000 mm,
	W =-180.000 deg,	P =   0.000 deg,	R =    90.000 deg
};
P[7159]{
   GP1:
	UF : 1, UT : 4,		CONFIG : 'N U T, 0, 0, 0',
	X =  22.000  mm,	Y =  148.000  mm,	Z =   15.000 mm,
	W =-180.000 deg,	P =   0.000 deg,	R =    90.000 deg
};
P[7160]{
   GP1:
	UF : 1, UT : 4,		CONFIG : 'N U T, 0, 0, 0',
	X =  22.000  mm,	Y =  148.000  mm,	Z =   -1.000 mm,
	W =-180.000 deg,	P =   0.000 deg,	R =    90.000 deg
};
P[7161]{
   GP1:
	UF : 1, UT : 4,		CONFIG : 'N U T, 0, 0, 0',
	X =  22.000  mm,	Y =  148.000  mm,	Z =   15.000 mm,
	W =-180.000 deg,	P =   0.000 deg,	R =    90.000 deg
};
P[7162]{
   GP1:
	UF : 1, UT : 4,		CONFIG : 'N U T, 0, 0, 0',
	X =  25.000  mm,	Y =  148.000  mm,	Z =   15.000 mm,
	W =-180.000 deg,	P =   0.000 deg,	R =    90.000 deg
};
P[7163]{
   GP1:
	UF : 1, UT : 4,		CONFIG : 'N U T, 0, 0, 0',
	X =  25.000  mm,	Y =  148.000  mm,	Z =   -1.000 mm,
	W =-180.000 deg,	P =   0.000 deg,	R =    90.000 deg
};
P[7164]{
   GP1:
	UF : 1, UT : 4,		CONFIG : 'N U T, 0, 0, 0',
	X =  25.000  mm,	Y =  148.000  mm,	Z =   15.000 mm,
	W =-180.000 deg,	P =   0.000 deg,	R =    90.000 deg
};
P[7165]{
   GP1:
	UF : 1, UT : 4,		CONFIG : 'N U T, 0, 0, 0',
	X =  28.000  mm,	Y =  148.000  mm,	Z =   15.000 mm,
	W =-180.000 deg,	P =   0.000 deg,	R =    90.000 deg
};
P[7166]{
   GP1:
	UF : 1, UT : 4,		CONFIG : 'N U T, 0, 0, 0',
	X =  28.000  mm,	Y =  148.000  mm,	Z =   -1.000 mm,
	W =-180.000 deg,	P =   0.000 deg,	R =    90.000 deg
};
P[7167]{
   GP1:
	UF : 1, UT : 4,		CONFIG : 'N U T, 0, 0, 0',
	X =  28.000  mm,	Y =  148.000  mm,	Z =   15.000 mm,
	W =-180.000 deg,	P =   0.000 deg,	R =    90.000 deg
};
P[7168]{
   GP1:
	UF : 1, UT : 4,		CONFIG : 'N U T, 0, 0, 0',
	X =  31.000  mm,	Y =  148.000  mm,	Z =   15.000 mm,
	W =-180.000 deg,	P =   0.000 deg,	R =    90.000 deg
};
P[7169]{
   GP1:
	UF : 1, UT : 4,		CONFIG : 'N U T, 0, 0, 0',
	X =  31.000  mm,	Y =  148.000  mm,	Z =   -1.000 mm,
	W =-180.000 deg,	P =   0.000 deg,	R =    90.000 deg
};
P[7170]{
   GP1:
	UF : 1, UT : 4,		CONFIG : 'N U T, 0, 0, 0',
	X =  31.000  mm,	Y =  148.000  mm,	Z =   15.000 mm,
	W =-180.000 deg,	P =   0.000 deg,	R =    90.000 deg
};
P[7171]{
   GP1:
	UF : 1, UT : 4,		CONFIG : 'N U T, 0, 0, 0',
	X =  34.000  mm,	Y =  148.000  mm,	Z =   15.000 mm,
	W =-180.000 deg,	P =   0.000 deg,	R =    90.000 deg
};
P[7172]{
   GP1:
	UF : 1, UT : 4,		CONFIG : 'N U T, 0, 0, 0',
	X =  34.000  mm,	Y =  148.000  mm,	Z =   -1.000 mm,
	W =-180.000 deg,	P =   0.000 deg,	R =    90.000 deg
};
P[7173]{
   GP1:
	UF : 1, UT : 4,		CONFIG : 'N U T, 0, 0, 0',
	X =  34.000  mm,	Y =  148.000  mm,	Z =   15.000 mm,
	W =-180.000 deg,	P =   0.000 deg,	R =    90.000 deg
};
P[7174]{
   GP1:
	UF : 1, UT : 4,		CONFIG : 'N U T, 0, 0, 0',
	X =  37.000  mm,	Y =  148.000  mm,	Z =   15.000 mm,
	W =-180.000 deg,	P =   0.000 deg,	R =    90.000 deg
};
P[7175]{
   GP1:
	UF : 1, UT : 4,		CONFIG : 'N U T, 0, 0, 0',
	X =  37.000  mm,	Y =  148.000  mm,	Z =   -1.000 mm,
	W =-180.000 deg,	P =   0.000 deg,	R =    90.000 deg
};
P[7176]{
   GP1:
	UF : 1, UT : 4,		CONFIG : 'N U T, 0, 0, 0',
	X =  37.000  mm,	Y =  148.000  mm,	Z =   15.000 mm,
	W =-180.000 deg,	P =   0.000 deg,	R =    90.000 deg
};
P[7177]{
   GP1:
	UF : 1, UT : 4,		CONFIG : 'N U T, 0, 0, 0',
	X =  40.000  mm,	Y =  148.000  mm,	Z =   15.000 mm,
	W =-180.000 deg,	P =   0.000 deg,	R =    90.000 deg
};
P[7178]{
   GP1:
	UF : 1, UT : 4,		CONFIG : 'N U T, 0, 0, 0',
	X =  40.000  mm,	Y =  148.000  mm,	Z =   -1.000 mm,
	W =-180.000 deg,	P =   0.000 deg,	R =    90.000 deg
};
P[7179]{
   GP1:
	UF : 1, UT : 4,		CONFIG : 'N U T, 0, 0, 0',
	X =  40.000  mm,	Y =  148.000  mm,	Z =   15.000 mm,
	W =-180.000 deg,	P =   0.000 deg,	R =    90.000 deg
};
P[7180]{
   GP1:
	UF : 1, UT : 4,		CONFIG : 'N U T, 0, 0, 0',
	X =  43.000  mm,	Y =  148.000  mm,	Z =   15.000 mm,
	W =-180.000 deg,	P =   0.000 deg,	R =    90.000 deg
};
P[7181]{
   GP1:
	UF : 1, UT : 4,		CONFIG : 'N U T, 0, 0, 0',
	X =  43.000  mm,	Y =  148.000  mm,	Z =   -1.000 mm,
	W =-180.000 deg,	P =   0.000 deg,	R =    90.000 deg
};
P[7182]{
   GP1:
	UF : 1, UT : 4,		CONFIG : 'N U T, 0, 0, 0',
	X =  43.000  mm,	Y =  148.000  mm,	Z =   15.000 mm,
	W =-180.000 deg,	P =   0.000 deg,	R =    90.000 deg
};
P[7183]{
   GP1:
	UF : 1, UT : 4,		CONFIG : 'N U T, 0, 0, 0',
	X =  46.000  mm,	Y =  148.000  mm,	Z =   15.000 mm,
	W =-180.000 deg,	P =   0.000 deg,	R =    90.000 deg
};
P[7184]{
   GP1:
	UF : 1, UT : 4,		CONFIG : 'N U T, 0, 0, 0',
	X =  46.000  mm,	Y =  148.000  mm,	Z =   -1.000 mm,
	W =-180.000 deg,	P =   0.000 deg,	R =    90.000 deg
};
P[7185]{
   GP1:
	UF : 1, UT : 4,		CONFIG : 'N U T, 0, 0, 0',
	X =  46.000  mm,	Y =  148.000  mm,	Z =   15.000 mm,
	W =-180.000 deg,	P =   0.000 deg,	R =    90.000 deg
};
P[7186]{
   GP1:
	UF : 1, UT : 4,		CONFIG : 'N U T, 0, 0, 0',
	X =  49.000  mm,	Y =  148.000  mm,	Z =   15.000 mm,
	W =-180.000 deg,	P =   0.000 deg,	R =    90.000 deg
};
P[7187]{
   GP1:
	UF : 1, UT : 4,		CONFIG : 'N U T, 0, 0, 0',
	X =  49.000  mm,	Y =  148.000  mm,	Z =   -1.000 mm,
	W =-180.000 deg,	P =   0.000 deg,	R =    90.000 deg
};
P[7188]{
   GP1:
	UF : 1, UT : 4,		CONFIG : 'N U T, 0, 0, 0',
	X =  49.000  mm,	Y =  148.000  mm,	Z =   15.000 mm,
	W =-180.000 deg,	P =   0.000 deg,	R =    90.000 deg
};
P[7189]{
   GP1:
	UF : 1, UT : 4,		CONFIG : 'N U T, 0, 0, 0',
	X =  52.000  mm,	Y =  148.000  mm,	Z =   15.000 mm,
	W =-180.000 deg,	P =   0.000 deg,	R =    90.000 deg
};
P[7190]{
   GP1:
	UF : 1, UT : 4,		CONFIG : 'N U T, 0, 0, 0',
	X =  52.000  mm,	Y =  148.000  mm,	Z =   -1.000 mm,
	W =-180.000 deg,	P =   0.000 deg,	R =    90.000 deg
};
P[7191]{
   GP1:
	UF : 1, UT : 4,		CONFIG : 'N U T, 0, 0, 0',
	X =  52.000  mm,	Y =  148.000  mm,	Z =   15.000 mm,
	W =-180.000 deg,	P =   0.000 deg,	R =    90.000 deg
};
P[7192]{
   GP1:
	UF : 1, UT : 4,		CONFIG : 'N U T, 0, 0, 0',
	X =  55.000  mm,	Y =  148.000  mm,	Z =   15.000 mm,
	W =-180.000 deg,	P =   0.000 deg,	R =    90.000 deg
};
P[7193]{
   GP1:
	UF : 1, UT : 4,		CONFIG : 'N U T, 0, 0, 0',
	X =  55.000  mm,	Y =  148.000  mm,	Z =   -1.000 mm,
	W =-180.000 deg,	P =   0.000 deg,	R =    90.000 deg
};
P[7194]{
   GP1:
	UF : 1, UT : 4,		CONFIG : 'N U T, 0, 0, 0',
	X =  55.000  mm,	Y =  148.000  mm,	Z =   15.000 mm,
	W =-180.000 deg,	P =   0.000 deg,	R =    90.000 deg
};
P[7195]{
   GP1:
	UF : 1, UT : 4,		CONFIG : 'N U T, 0, 0, 0',
	X =  58.000  mm,	Y =  148.000  mm,	Z =   15.000 mm,
	W =-180.000 deg,	P =   0.000 deg,	R =    90.000 deg
};
P[7196]{
   GP1:
	UF : 1, UT : 4,		CONFIG : 'N U T, 0, 0, 0',
	X =  58.000  mm,	Y =  148.000  mm,	Z =   -1.000 mm,
	W =-180.000 deg,	P =   0.000 deg,	R =    90.000 deg
};
P[7197]{
   GP1:
	UF : 1, UT : 4,		CONFIG : 'N U T, 0, 0, 0',
	X =  58.000  mm,	Y =  148.000  mm,	Z =   15.000 mm,
	W =-180.000 deg,	P =   0.000 deg,	R =    90.000 deg
};
P[7198]{
   GP1:
	UF : 1, UT : 4,		CONFIG : 'N U T, 0, 0, 0',
	X =  61.000  mm,	Y =  148.000  mm,	Z =   15.000 mm,
	W =-180.000 deg,	P =   0.000 deg,	R =    90.000 deg
};
P[7199]{
   GP1:
	UF : 1, UT : 4,		CONFIG : 'N U T, 0, 0, 0',
	X =  61.000  mm,	Y =  148.000  mm,	Z =   -1.000 mm,
	W =-180.000 deg,	P =   0.000 deg,	R =    90.000 deg
};
P[7200]{
   GP1:
	UF : 1, UT : 4,		CONFIG : 'N U T, 0, 0, 0',
	X =  61.000  mm,	Y =  148.000  mm,	Z =   15.000 mm,
	W =-180.000 deg,	P =   0.000 deg,	R =    90.000 deg
};
P[7222]{
   GP1:
	UF : 1, UT : 4,		CONFIG : 'N U T, 0, 0, 0',
	X =  124.000  mm,	Y =  148.000  mm,	Z =   15.000 mm,
	W =-180.000 deg,	P =   0.000 deg,	R =    90.000 deg
};
P[7223]{
   GP1:
	UF : 1, UT : 4,		CONFIG : 'N U T, 0, 0, 0',
	X =  124.000  mm,	Y =  148.000  mm,	Z =   -1.000 mm,
	W =-180.000 deg,	P =   0.000 deg,	R =    90.000 deg
};
P[7224]{
   GP1:
	UF : 1, UT : 4,		CONFIG : 'N U T, 0, 0, 0',
	X =  124.000  mm,	Y =  148.000  mm,	Z =   15.000 mm,
	W =-180.000 deg,	P =   0.000 deg,	R =    90.000 deg
};
P[7225]{
   GP1:
	UF : 1, UT : 4,		CONFIG : 'N U T, 0, 0, 0',
	X =  127.000  mm,	Y =  148.000  mm,	Z =   15.000 mm,
	W =-180.000 deg,	P =   0.000 deg,	R =    90.000 deg
};
P[7226]{
   GP1:
	UF : 1, UT : 4,		CONFIG : 'N U T, 0, 0, 0',
	X =  127.000  mm,	Y =  148.000  mm,	Z =   -1.000 mm,
	W =-180.000 deg,	P =   0.000 deg,	R =    90.000 deg
};
P[7227]{
   GP1:
	UF : 1, UT : 4,		CONFIG : 'N U T, 0, 0, 0',
	X =  127.000  mm,	Y =  148.000  mm,	Z =   15.000 mm,
	W =-180.000 deg,	P =   0.000 deg,	R =    90.000 deg
};
P[7240]{
   GP1:
	UF : 1, UT : 4,		CONFIG : 'N U T, 0, 0, 0',
	X =  142.000  mm,	Y =  148.000  mm,	Z =   15.000 mm,
	W =-180.000 deg,	P =   0.000 deg,	R =    90.000 deg
};
P[7241]{
   GP1:
	UF : 1, UT : 4,		CONFIG : 'N U T, 0, 0, 0',
	X =  142.000  mm,	Y =  148.000  mm,	Z =   -1.000 mm,
	W =-180.000 deg,	P =   0.000 deg,	R =    90.000 deg
};
P[7242]{
   GP1:
	UF : 1, UT : 4,		CONFIG : 'N U T, 0, 0, 0',
	X =  142.000  mm,	Y =  148.000  mm,	Z =   15.000 mm,
	W =-180.000 deg,	P =   0.000 deg,	R =    90.000 deg
};
P[7243]{
   GP1:
	UF : 1, UT : 4,		CONFIG : 'N U T, 0, 0, 0',
	X =  145.000  mm,	Y =  148.000  mm,	Z =   15.000 mm,
	W =-180.000 deg,	P =   0.000 deg,	R =    90.000 deg
};
P[7244]{
   GP1:
	UF : 1, UT : 4,		CONFIG : 'N U T, 0, 0, 0',
	X =  145.000  mm,	Y =  148.000  mm,	Z =   -1.000 mm,
	W =-180.000 deg,	P =   0.000 deg,	R =    90.000 deg
};
P[7245]{
   GP1:
	UF : 1, UT : 4,		CONFIG : 'N U T, 0, 0, 0',
	X =  145.000  mm,	Y =  148.000  mm,	Z =   15.000 mm,
	W =-180.000 deg,	P =   0.000 deg,	R =    90.000 deg
};
P[7246]{
   GP1:
	UF : 1, UT : 4,		CONFIG : 'N U T, 0, 0, 0',
	X =  148.000  mm,	Y =  148.000  mm,	Z =   15.000 mm,
	W =-180.000 deg,	P =   0.000 deg,	R =    90.000 deg
};
P[7247]{
   GP1:
	UF : 1, UT : 4,		CONFIG : 'N U T, 0, 0, 0',
	X =  148.000  mm,	Y =  148.000  mm,	Z =   -1.000 mm,
	W =-180.000 deg,	P =   0.000 deg,	R =    90.000 deg
};
P[7248]{
   GP1:
	UF : 1, UT : 4,		CONFIG : 'N U T, 0, 0, 0',
	X =  148.000  mm,	Y =  148.000  mm,	Z =   15.000 mm,
	W =-180.000 deg,	P =   0.000 deg,	R =    90.000 deg
};
P[7249]{
   GP1:
	UF : 1, UT : 4,		CONFIG : 'N U T, 0, 0, 0',
	X =  151.000  mm,	Y =  148.000  mm,	Z =   15.000 mm,
	W =-180.000 deg,	P =   0.000 deg,	R =    90.000 deg
};
P[7250]{
   GP1:
	UF : 1, UT : 4,		CONFIG : 'N U T, 0, 0, 0',
	X =  151.000  mm,	Y =  148.000  mm,	Z =   -1.000 mm,
	W =-180.000 deg,	P =   0.000 deg,	R =    90.000 deg
};
P[7251]{
   GP1:
	UF : 1, UT : 4,		CONFIG : 'N U T, 0, 0, 0',
	X =  151.000  mm,	Y =  148.000  mm,	Z =   15.000 mm,
	W =-180.000 deg,	P =   0.000 deg,	R =    90.000 deg
};
P[7264]{
   GP1:
	UF : 1, UT : 4,		CONFIG : 'N U T, 0, 0, 0',
	X =  22.000  mm,	Y =  151.000  mm,	Z =   15.000 mm,
	W =-180.000 deg,	P =   0.000 deg,	R =    90.000 deg
};
P[7265]{
   GP1:
	UF : 1, UT : 4,		CONFIG : 'N U T, 0, 0, 0',
	X =  22.000  mm,	Y =  151.000  mm,	Z =   -1.000 mm,
	W =-180.000 deg,	P =   0.000 deg,	R =    90.000 deg
};
P[7266]{
   GP1:
	UF : 1, UT : 4,		CONFIG : 'N U T, 0, 0, 0',
	X =  22.000  mm,	Y =  151.000  mm,	Z =   15.000 mm,
	W =-180.000 deg,	P =   0.000 deg,	R =    90.000 deg
};
P[7267]{
   GP1:
	UF : 1, UT : 4,		CONFIG : 'N U T, 0, 0, 0',
	X =  25.000  mm,	Y =  151.000  mm,	Z =   15.000 mm,
	W =-180.000 deg,	P =   0.000 deg,	R =    90.000 deg
};
P[7268]{
   GP1:
	UF : 1, UT : 4,		CONFIG : 'N U T, 0, 0, 0',
	X =  25.000  mm,	Y =  151.000  mm,	Z =   -1.000 mm,
	W =-180.000 deg,	P =   0.000 deg,	R =    90.000 deg
};
P[7269]{
   GP1:
	UF : 1, UT : 4,		CONFIG : 'N U T, 0, 0, 0',
	X =  25.000  mm,	Y =  151.000  mm,	Z =   15.000 mm,
	W =-180.000 deg,	P =   0.000 deg,	R =    90.000 deg
};
P[7270]{
   GP1:
	UF : 1, UT : 4,		CONFIG : 'N U T, 0, 0, 0',
	X =  28.000  mm,	Y =  151.000  mm,	Z =   15.000 mm,
	W =-180.000 deg,	P =   0.000 deg,	R =    90.000 deg
};
P[7271]{
   GP1:
	UF : 1, UT : 4,		CONFIG : 'N U T, 0, 0, 0',
	X =  28.000  mm,	Y =  151.000  mm,	Z =   -1.000 mm,
	W =-180.000 deg,	P =   0.000 deg,	R =    90.000 deg
};
P[7272]{
   GP1:
	UF : 1, UT : 4,		CONFIG : 'N U T, 0, 0, 0',
	X =  28.000  mm,	Y =  151.000  mm,	Z =   15.000 mm,
	W =-180.000 deg,	P =   0.000 deg,	R =    90.000 deg
};
P[7273]{
   GP1:
	UF : 1, UT : 4,		CONFIG : 'N U T, 0, 0, 0',
	X =  31.000  mm,	Y =  151.000  mm,	Z =   15.000 mm,
	W =-180.000 deg,	P =   0.000 deg,	R =    90.000 deg
};
P[7274]{
   GP1:
	UF : 1, UT : 4,		CONFIG : 'N U T, 0, 0, 0',
	X =  31.000  mm,	Y =  151.000  mm,	Z =   -1.000 mm,
	W =-180.000 deg,	P =   0.000 deg,	R =    90.000 deg
};
P[7275]{
   GP1:
	UF : 1, UT : 4,		CONFIG : 'N U T, 0, 0, 0',
	X =  31.000  mm,	Y =  151.000  mm,	Z =   15.000 mm,
	W =-180.000 deg,	P =   0.000 deg,	R =    90.000 deg
};
P[7276]{
   GP1:
	UF : 1, UT : 4,		CONFIG : 'N U T, 0, 0, 0',
	X =  34.000  mm,	Y =  151.000  mm,	Z =   15.000 mm,
	W =-180.000 deg,	P =   0.000 deg,	R =    90.000 deg
};
P[7277]{
   GP1:
	UF : 1, UT : 4,		CONFIG : 'N U T, 0, 0, 0',
	X =  34.000  mm,	Y =  151.000  mm,	Z =   -1.000 mm,
	W =-180.000 deg,	P =   0.000 deg,	R =    90.000 deg
};
P[7278]{
   GP1:
	UF : 1, UT : 4,		CONFIG : 'N U T, 0, 0, 0',
	X =  34.000  mm,	Y =  151.000  mm,	Z =   15.000 mm,
	W =-180.000 deg,	P =   0.000 deg,	R =    90.000 deg
};
P[7279]{
   GP1:
	UF : 1, UT : 4,		CONFIG : 'N U T, 0, 0, 0',
	X =  37.000  mm,	Y =  151.000  mm,	Z =   15.000 mm,
	W =-180.000 deg,	P =   0.000 deg,	R =    90.000 deg
};
P[7280]{
   GP1:
	UF : 1, UT : 4,		CONFIG : 'N U T, 0, 0, 0',
	X =  37.000  mm,	Y =  151.000  mm,	Z =   -1.000 mm,
	W =-180.000 deg,	P =   0.000 deg,	R =    90.000 deg
};
P[7281]{
   GP1:
	UF : 1, UT : 4,		CONFIG : 'N U T, 0, 0, 0',
	X =  37.000  mm,	Y =  151.000  mm,	Z =   15.000 mm,
	W =-180.000 deg,	P =   0.000 deg,	R =    90.000 deg
};
P[7282]{
   GP1:
	UF : 1, UT : 4,		CONFIG : 'N U T, 0, 0, 0',
	X =  40.000  mm,	Y =  151.000  mm,	Z =   15.000 mm,
	W =-180.000 deg,	P =   0.000 deg,	R =    90.000 deg
};
P[7283]{
   GP1:
	UF : 1, UT : 4,		CONFIG : 'N U T, 0, 0, 0',
	X =  40.000  mm,	Y =  151.000  mm,	Z =   -1.000 mm,
	W =-180.000 deg,	P =   0.000 deg,	R =    90.000 deg
};
P[7284]{
   GP1:
	UF : 1, UT : 4,		CONFIG : 'N U T, 0, 0, 0',
	X =  40.000  mm,	Y =  151.000  mm,	Z =   15.000 mm,
	W =-180.000 deg,	P =   0.000 deg,	R =    90.000 deg
};
P[7285]{
   GP1:
	UF : 1, UT : 4,		CONFIG : 'N U T, 0, 0, 0',
	X =  43.000  mm,	Y =  151.000  mm,	Z =   15.000 mm,
	W =-180.000 deg,	P =   0.000 deg,	R =    90.000 deg
};
P[7286]{
   GP1:
	UF : 1, UT : 4,		CONFIG : 'N U T, 0, 0, 0',
	X =  43.000  mm,	Y =  151.000  mm,	Z =   -1.000 mm,
	W =-180.000 deg,	P =   0.000 deg,	R =    90.000 deg
};
P[7287]{
   GP1:
	UF : 1, UT : 4,		CONFIG : 'N U T, 0, 0, 0',
	X =  43.000  mm,	Y =  151.000  mm,	Z =   15.000 mm,
	W =-180.000 deg,	P =   0.000 deg,	R =    90.000 deg
};
P[7288]{
   GP1:
	UF : 1, UT : 4,		CONFIG : 'N U T, 0, 0, 0',
	X =  46.000  mm,	Y =  151.000  mm,	Z =   15.000 mm,
	W =-180.000 deg,	P =   0.000 deg,	R =    90.000 deg
};
P[7289]{
   GP1:
	UF : 1, UT : 4,		CONFIG : 'N U T, 0, 0, 0',
	X =  46.000  mm,	Y =  151.000  mm,	Z =   -1.000 mm,
	W =-180.000 deg,	P =   0.000 deg,	R =    90.000 deg
};
P[7290]{
   GP1:
	UF : 1, UT : 4,		CONFIG : 'N U T, 0, 0, 0',
	X =  46.000  mm,	Y =  151.000  mm,	Z =   15.000 mm,
	W =-180.000 deg,	P =   0.000 deg,	R =    90.000 deg
};
P[7291]{
   GP1:
	UF : 1, UT : 4,		CONFIG : 'N U T, 0, 0, 0',
	X =  49.000  mm,	Y =  151.000  mm,	Z =   15.000 mm,
	W =-180.000 deg,	P =   0.000 deg,	R =    90.000 deg
};
P[7292]{
   GP1:
	UF : 1, UT : 4,		CONFIG : 'N U T, 0, 0, 0',
	X =  49.000  mm,	Y =  151.000  mm,	Z =   -1.000 mm,
	W =-180.000 deg,	P =   0.000 deg,	R =    90.000 deg
};
P[7293]{
   GP1:
	UF : 1, UT : 4,		CONFIG : 'N U T, 0, 0, 0',
	X =  49.000  mm,	Y =  151.000  mm,	Z =   15.000 mm,
	W =-180.000 deg,	P =   0.000 deg,	R =    90.000 deg
};
P[7294]{
   GP1:
	UF : 1, UT : 4,		CONFIG : 'N U T, 0, 0, 0',
	X =  52.000  mm,	Y =  151.000  mm,	Z =   15.000 mm,
	W =-180.000 deg,	P =   0.000 deg,	R =    90.000 deg
};
P[7295]{
   GP1:
	UF : 1, UT : 4,		CONFIG : 'N U T, 0, 0, 0',
	X =  52.000  mm,	Y =  151.000  mm,	Z =   -1.000 mm,
	W =-180.000 deg,	P =   0.000 deg,	R =    90.000 deg
};
P[7296]{
   GP1:
	UF : 1, UT : 4,		CONFIG : 'N U T, 0, 0, 0',
	X =  52.000  mm,	Y =  151.000  mm,	Z =   15.000 mm,
	W =-180.000 deg,	P =   0.000 deg,	R =    90.000 deg
};
P[7297]{
   GP1:
	UF : 1, UT : 4,		CONFIG : 'N U T, 0, 0, 0',
	X =  55.000  mm,	Y =  151.000  mm,	Z =   15.000 mm,
	W =-180.000 deg,	P =   0.000 deg,	R =    90.000 deg
};
P[7298]{
   GP1:
	UF : 1, UT : 4,		CONFIG : 'N U T, 0, 0, 0',
	X =  55.000  mm,	Y =  151.000  mm,	Z =   -1.000 mm,
	W =-180.000 deg,	P =   0.000 deg,	R =    90.000 deg
};
P[7299]{
   GP1:
	UF : 1, UT : 4,		CONFIG : 'N U T, 0, 0, 0',
	X =  55.000  mm,	Y =  151.000  mm,	Z =   15.000 mm,
	W =-180.000 deg,	P =   0.000 deg,	R =    90.000 deg
};
P[7300]{
   GP1:
	UF : 1, UT : 4,		CONFIG : 'N U T, 0, 0, 0',
	X =  58.000  mm,	Y =  151.000  mm,	Z =   15.000 mm,
	W =-180.000 deg,	P =   0.000 deg,	R =    90.000 deg
};
P[7301]{
   GP1:
	UF : 1, UT : 4,		CONFIG : 'N U T, 0, 0, 0',
	X =  58.000  mm,	Y =  151.000  mm,	Z =   -1.000 mm,
	W =-180.000 deg,	P =   0.000 deg,	R =    90.000 deg
};
P[7302]{
   GP1:
	UF : 1, UT : 4,		CONFIG : 'N U T, 0, 0, 0',
	X =  58.000  mm,	Y =  151.000  mm,	Z =   15.000 mm,
	W =-180.000 deg,	P =   0.000 deg,	R =    90.000 deg
};
P[7303]{
   GP1:
	UF : 1, UT : 4,		CONFIG : 'N U T, 0, 0, 0',
	X =  61.000  mm,	Y =  151.000  mm,	Z =   15.000 mm,
	W =-180.000 deg,	P =   0.000 deg,	R =    90.000 deg
};
P[7304]{
   GP1:
	UF : 1, UT : 4,		CONFIG : 'N U T, 0, 0, 0',
	X =  61.000  mm,	Y =  151.000  mm,	Z =   -1.000 mm,
	W =-180.000 deg,	P =   0.000 deg,	R =    90.000 deg
};
P[7305]{
   GP1:
	UF : 1, UT : 4,		CONFIG : 'N U T, 0, 0, 0',
	X =  61.000  mm,	Y =  151.000  mm,	Z =   15.000 mm,
	W =-180.000 deg,	P =   0.000 deg,	R =    90.000 deg
};
P[7330]{
   GP1:
	UF : 1, UT : 4,		CONFIG : 'N U T, 0, 0, 0',
	X =  127.000  mm,	Y =  151.000  mm,	Z =   15.000 mm,
	W =-180.000 deg,	P =   0.000 deg,	R =    90.000 deg
};
P[7331]{
   GP1:
	UF : 1, UT : 4,		CONFIG : 'N U T, 0, 0, 0',
	X =  127.000  mm,	Y =  151.000  mm,	Z =   -1.000 mm,
	W =-180.000 deg,	P =   0.000 deg,	R =    90.000 deg
};
P[7332]{
   GP1:
	UF : 1, UT : 4,		CONFIG : 'N U T, 0, 0, 0',
	X =  127.000  mm,	Y =  151.000  mm,	Z =   15.000 mm,
	W =-180.000 deg,	P =   0.000 deg,	R =    90.000 deg
};
P[7348]{
   GP1:
	UF : 1, UT : 4,		CONFIG : 'N U T, 0, 0, 0',
	X =  145.000  mm,	Y =  151.000  mm,	Z =   15.000 mm,
	W =-180.000 deg,	P =   0.000 deg,	R =    90.000 deg
};
P[7349]{
   GP1:
	UF : 1, UT : 4,		CONFIG : 'N U T, 0, 0, 0',
	X =  145.000  mm,	Y =  151.000  mm,	Z =   -1.000 mm,
	W =-180.000 deg,	P =   0.000 deg,	R =    90.000 deg
};
P[7350]{
   GP1:
	UF : 1, UT : 4,		CONFIG : 'N U T, 0, 0, 0',
	X =  145.000  mm,	Y =  151.000  mm,	Z =   15.000 mm,
	W =-180.000 deg,	P =   0.000 deg,	R =    90.000 deg
};
P[7351]{
   GP1:
	UF : 1, UT : 4,		CONFIG : 'N U T, 0, 0, 0',
	X =  148.000  mm,	Y =  151.000  mm,	Z =   15.000 mm,
	W =-180.000 deg,	P =   0.000 deg,	R =    90.000 deg
};
P[7352]{
   GP1:
	UF : 1, UT : 4,		CONFIG : 'N U T, 0, 0, 0',
	X =  148.000  mm,	Y =  151.000  mm,	Z =   -1.000 mm,
	W =-180.000 deg,	P =   0.000 deg,	R =    90.000 deg
};
P[7353]{
   GP1:
	UF : 1, UT : 4,		CONFIG : 'N U T, 0, 0, 0',
	X =  148.000  mm,	Y =  151.000  mm,	Z =   15.000 mm,
	W =-180.000 deg,	P =   0.000 deg,	R =    90.000 deg
};
P[7354]{
   GP1:
	UF : 1, UT : 4,		CONFIG : 'N U T, 0, 0, 0',
	X =  151.000  mm,	Y =  151.000  mm,	Z =   15.000 mm,
	W =-180.000 deg,	P =   0.000 deg,	R =    90.000 deg
};
P[7355]{
   GP1:
	UF : 1, UT : 4,		CONFIG : 'N U T, 0, 0, 0',
	X =  151.000  mm,	Y =  151.000  mm,	Z =   -1.000 mm,
	W =-180.000 deg,	P =   0.000 deg,	R =    90.000 deg
};
P[7356]{
   GP1:
	UF : 1, UT : 4,		CONFIG : 'N U T, 0, 0, 0',
	X =  151.000  mm,	Y =  151.000  mm,	Z =   15.000 mm,
	W =-180.000 deg,	P =   0.000 deg,	R =    90.000 deg
};
P[7369]{
   GP1:
	UF : 1, UT : 4,		CONFIG : 'N U T, 0, 0, 0',
	X =  22.000  mm,	Y =  154.000  mm,	Z =   15.000 mm,
	W =-180.000 deg,	P =   0.000 deg,	R =    90.000 deg
};
P[7370]{
   GP1:
	UF : 1, UT : 4,		CONFIG : 'N U T, 0, 0, 0',
	X =  22.000  mm,	Y =  154.000  mm,	Z =   -1.000 mm,
	W =-180.000 deg,	P =   0.000 deg,	R =    90.000 deg
};
P[7371]{
   GP1:
	UF : 1, UT : 4,		CONFIG : 'N U T, 0, 0, 0',
	X =  22.000  mm,	Y =  154.000  mm,	Z =   15.000 mm,
	W =-180.000 deg,	P =   0.000 deg,	R =    90.000 deg
};
P[7372]{
   GP1:
	UF : 1, UT : 4,		CONFIG : 'N U T, 0, 0, 0',
	X =  25.000  mm,	Y =  154.000  mm,	Z =   15.000 mm,
	W =-180.000 deg,	P =   0.000 deg,	R =    90.000 deg
};
P[7373]{
   GP1:
	UF : 1, UT : 4,		CONFIG : 'N U T, 0, 0, 0',
	X =  25.000  mm,	Y =  154.000  mm,	Z =   -1.000 mm,
	W =-180.000 deg,	P =   0.000 deg,	R =    90.000 deg
};
P[7374]{
   GP1:
	UF : 1, UT : 4,		CONFIG : 'N U T, 0, 0, 0',
	X =  25.000  mm,	Y =  154.000  mm,	Z =   15.000 mm,
	W =-180.000 deg,	P =   0.000 deg,	R =    90.000 deg
};
P[7375]{
   GP1:
	UF : 1, UT : 4,		CONFIG : 'N U T, 0, 0, 0',
	X =  28.000  mm,	Y =  154.000  mm,	Z =   15.000 mm,
	W =-180.000 deg,	P =   0.000 deg,	R =    90.000 deg
};
P[7376]{
   GP1:
	UF : 1, UT : 4,		CONFIG : 'N U T, 0, 0, 0',
	X =  28.000  mm,	Y =  154.000  mm,	Z =   -1.000 mm,
	W =-180.000 deg,	P =   0.000 deg,	R =    90.000 deg
};
P[7377]{
   GP1:
	UF : 1, UT : 4,		CONFIG : 'N U T, 0, 0, 0',
	X =  28.000  mm,	Y =  154.000  mm,	Z =   15.000 mm,
	W =-180.000 deg,	P =   0.000 deg,	R =    90.000 deg
};
P[7378]{
   GP1:
	UF : 1, UT : 4,		CONFIG : 'N U T, 0, 0, 0',
	X =  31.000  mm,	Y =  154.000  mm,	Z =   15.000 mm,
	W =-180.000 deg,	P =   0.000 deg,	R =    90.000 deg
};
P[7379]{
   GP1:
	UF : 1, UT : 4,		CONFIG : 'N U T, 0, 0, 0',
	X =  31.000  mm,	Y =  154.000  mm,	Z =   -1.000 mm,
	W =-180.000 deg,	P =   0.000 deg,	R =    90.000 deg
};
P[7380]{
   GP1:
	UF : 1, UT : 4,		CONFIG : 'N U T, 0, 0, 0',
	X =  31.000  mm,	Y =  154.000  mm,	Z =   15.000 mm,
	W =-180.000 deg,	P =   0.000 deg,	R =    90.000 deg
};
P[7381]{
   GP1:
	UF : 1, UT : 4,		CONFIG : 'N U T, 0, 0, 0',
	X =  34.000  mm,	Y =  154.000  mm,	Z =   15.000 mm,
	W =-180.000 deg,	P =   0.000 deg,	R =    90.000 deg
};
P[7382]{
   GP1:
	UF : 1, UT : 4,		CONFIG : 'N U T, 0, 0, 0',
	X =  34.000  mm,	Y =  154.000  mm,	Z =   -1.000 mm,
	W =-180.000 deg,	P =   0.000 deg,	R =    90.000 deg
};
P[7383]{
   GP1:
	UF : 1, UT : 4,		CONFIG : 'N U T, 0, 0, 0',
	X =  34.000  mm,	Y =  154.000  mm,	Z =   15.000 mm,
	W =-180.000 deg,	P =   0.000 deg,	R =    90.000 deg
};
P[7384]{
   GP1:
	UF : 1, UT : 4,		CONFIG : 'N U T, 0, 0, 0',
	X =  37.000  mm,	Y =  154.000  mm,	Z =   15.000 mm,
	W =-180.000 deg,	P =   0.000 deg,	R =    90.000 deg
};
P[7385]{
   GP1:
	UF : 1, UT : 4,		CONFIG : 'N U T, 0, 0, 0',
	X =  37.000  mm,	Y =  154.000  mm,	Z =   -1.000 mm,
	W =-180.000 deg,	P =   0.000 deg,	R =    90.000 deg
};
P[7386]{
   GP1:
	UF : 1, UT : 4,		CONFIG : 'N U T, 0, 0, 0',
	X =  37.000  mm,	Y =  154.000  mm,	Z =   15.000 mm,
	W =-180.000 deg,	P =   0.000 deg,	R =    90.000 deg
};
P[7387]{
   GP1:
	UF : 1, UT : 4,		CONFIG : 'N U T, 0, 0, 0',
	X =  40.000  mm,	Y =  154.000  mm,	Z =   15.000 mm,
	W =-180.000 deg,	P =   0.000 deg,	R =    90.000 deg
};
P[7388]{
   GP1:
	UF : 1, UT : 4,		CONFIG : 'N U T, 0, 0, 0',
	X =  40.000  mm,	Y =  154.000  mm,	Z =   -1.000 mm,
	W =-180.000 deg,	P =   0.000 deg,	R =    90.000 deg
};
P[7389]{
   GP1:
	UF : 1, UT : 4,		CONFIG : 'N U T, 0, 0, 0',
	X =  40.000  mm,	Y =  154.000  mm,	Z =   15.000 mm,
	W =-180.000 deg,	P =   0.000 deg,	R =    90.000 deg
};
P[7390]{
   GP1:
	UF : 1, UT : 4,		CONFIG : 'N U T, 0, 0, 0',
	X =  43.000  mm,	Y =  154.000  mm,	Z =   15.000 mm,
	W =-180.000 deg,	P =   0.000 deg,	R =    90.000 deg
};
P[7391]{
   GP1:
	UF : 1, UT : 4,		CONFIG : 'N U T, 0, 0, 0',
	X =  43.000  mm,	Y =  154.000  mm,	Z =   -1.000 mm,
	W =-180.000 deg,	P =   0.000 deg,	R =    90.000 deg
};
P[7392]{
   GP1:
	UF : 1, UT : 4,		CONFIG : 'N U T, 0, 0, 0',
	X =  43.000  mm,	Y =  154.000  mm,	Z =   15.000 mm,
	W =-180.000 deg,	P =   0.000 deg,	R =    90.000 deg
};
P[7393]{
   GP1:
	UF : 1, UT : 4,		CONFIG : 'N U T, 0, 0, 0',
	X =  46.000  mm,	Y =  154.000  mm,	Z =   15.000 mm,
	W =-180.000 deg,	P =   0.000 deg,	R =    90.000 deg
};
P[7394]{
   GP1:
	UF : 1, UT : 4,		CONFIG : 'N U T, 0, 0, 0',
	X =  46.000  mm,	Y =  154.000  mm,	Z =   -1.000 mm,
	W =-180.000 deg,	P =   0.000 deg,	R =    90.000 deg
};
P[7395]{
   GP1:
	UF : 1, UT : 4,		CONFIG : 'N U T, 0, 0, 0',
	X =  46.000  mm,	Y =  154.000  mm,	Z =   15.000 mm,
	W =-180.000 deg,	P =   0.000 deg,	R =    90.000 deg
};
P[7396]{
   GP1:
	UF : 1, UT : 4,		CONFIG : 'N U T, 0, 0, 0',
	X =  49.000  mm,	Y =  154.000  mm,	Z =   15.000 mm,
	W =-180.000 deg,	P =   0.000 deg,	R =    90.000 deg
};
P[7397]{
   GP1:
	UF : 1, UT : 4,		CONFIG : 'N U T, 0, 0, 0',
	X =  49.000  mm,	Y =  154.000  mm,	Z =   -1.000 mm,
	W =-180.000 deg,	P =   0.000 deg,	R =    90.000 deg
};
P[7398]{
   GP1:
	UF : 1, UT : 4,		CONFIG : 'N U T, 0, 0, 0',
	X =  49.000  mm,	Y =  154.000  mm,	Z =   15.000 mm,
	W =-180.000 deg,	P =   0.000 deg,	R =    90.000 deg
};
P[7399]{
   GP1:
	UF : 1, UT : 4,		CONFIG : 'N U T, 0, 0, 0',
	X =  52.000  mm,	Y =  154.000  mm,	Z =   15.000 mm,
	W =-180.000 deg,	P =   0.000 deg,	R =    90.000 deg
};
P[7400]{
   GP1:
	UF : 1, UT : 4,		CONFIG : 'N U T, 0, 0, 0',
	X =  52.000  mm,	Y =  154.000  mm,	Z =   -1.000 mm,
	W =-180.000 deg,	P =   0.000 deg,	R =    90.000 deg
};
P[7401]{
   GP1:
	UF : 1, UT : 4,		CONFIG : 'N U T, 0, 0, 0',
	X =  52.000  mm,	Y =  154.000  mm,	Z =   15.000 mm,
	W =-180.000 deg,	P =   0.000 deg,	R =    90.000 deg
};
P[7402]{
   GP1:
	UF : 1, UT : 4,		CONFIG : 'N U T, 0, 0, 0',
	X =  55.000  mm,	Y =  154.000  mm,	Z =   15.000 mm,
	W =-180.000 deg,	P =   0.000 deg,	R =    90.000 deg
};
P[7403]{
   GP1:
	UF : 1, UT : 4,		CONFIG : 'N U T, 0, 0, 0',
	X =  55.000  mm,	Y =  154.000  mm,	Z =   -1.000 mm,
	W =-180.000 deg,	P =   0.000 deg,	R =    90.000 deg
};
P[7404]{
   GP1:
	UF : 1, UT : 4,		CONFIG : 'N U T, 0, 0, 0',
	X =  55.000  mm,	Y =  154.000  mm,	Z =   15.000 mm,
	W =-180.000 deg,	P =   0.000 deg,	R =    90.000 deg
};
P[7405]{
   GP1:
	UF : 1, UT : 4,		CONFIG : 'N U T, 0, 0, 0',
	X =  58.000  mm,	Y =  154.000  mm,	Z =   15.000 mm,
	W =-180.000 deg,	P =   0.000 deg,	R =    90.000 deg
};
P[7406]{
   GP1:
	UF : 1, UT : 4,		CONFIG : 'N U T, 0, 0, 0',
	X =  58.000  mm,	Y =  154.000  mm,	Z =   -1.000 mm,
	W =-180.000 deg,	P =   0.000 deg,	R =    90.000 deg
};
P[7407]{
   GP1:
	UF : 1, UT : 4,		CONFIG : 'N U T, 0, 0, 0',
	X =  58.000  mm,	Y =  154.000  mm,	Z =   15.000 mm,
	W =-180.000 deg,	P =   0.000 deg,	R =    90.000 deg
};
P[7453]{
   GP1:
